// TwinCAT 3 PLC project xPPU_Lib
// Title: xPPU
// Company: Jan Wilch
// ProjectVersion: 1.0.0
// ProgramVersion: 3.1.4026.11
// libraries:
//   Tc2_Standard, * (Beckhoff Automation GmbH)
//   Tc2_System, * (Beckhoff Automation GmbH)
//   Tc3_Module, * (Beckhoff Automation GmbH)
//   [Resi4MPM], * (Jan Wilch)
// project tree:
//   03_ControlPrimitives/Carrier/Crane/ Crane_MoveBase.TcPOU, Crane_MoveToLSC.TcPOU, Crane_MoveToStack.TcPOU, Crane_MoveToStamp.TcPOU, Crane_PickPutBase.TcPOU, Crane_PickUpWP.TcPOU, Crane_PutDownWP.TcPOU
//   03_ControlPrimitives/Carrier/PickAlpha/ PicAlpha_MoveBase.TcPOU, PicAlpha_MoveToPos1.TcPOU, PicAlpha_MoveToPos2.TcPOU, PicAlpha_MoveToPos3.TcPOU, PicAlpha_MoveToPos4.TcPOU, PicAlpha_PickUpWP.TcPOU, PicAlpha_PutDownWP.TcPOU
//   03_ControlPrimitives/Conveyor/LSC/ LSC_MoveWorkpiece_Base.TcPOU, LSC_SearchWorkpiece.TcPOU, LSC_TransferWorkpieceTo_PAC.TcPOU, LSC_TransferWorkpieceTo_RampEnd.TcPOU, LSC_TransferWorkpieceTo_RampMid.TcPOU, LSC_TransferWorkpieceTo_RampStart.TcPOU
//   03_ControlPrimitives/Conveyor/PAC/ PAC_MoveWorkpiece_Base.TcPOU, PAC_TransferWorkpieceTo_PSEnd.TcPOU, PAC_TransferWorkpieceTo_PSStart.TcPOU, PAC_TransferWorkpieceTo_SSC.TcPOU
//   03_ControlPrimitives/Conveyor/RFC/ RFC_MoveWorkpiece_Base.TcPOU, RFC_TransferWorkpieceTo_LSC.TcPOU, RFC_TransferWorkpieceTo_PSEnd.TcPOU
//   03_ControlPrimitives/Conveyor/SSC/ SSC_MoveWorkpiece_Base.TcPOU, SSC_TransferWorkpieceTo_PSStart.TcPOU, SSC_TransferWorkpieceTo_RampEnd.TcPOU, SSC_TransferWorkpieceTo_RFC.TcPOU
//   03_ControlPrimitives/Generic/ Delay.TcPOU, ForceProcessVariable.TcPOU, IndicateActivity.TcPOU
//   03_ControlPrimitives/Stack/ Stack_ProvideWorkpiece.TcPOU
//   03_ControlPrimitives/Stamp/ Stamp_StampWorkpiece.TcPOU
//   04_HardwareObservation/ ObserveCrane.TcPOU, ObserveLSC.TcPOU, ObservePAC.TcPOU, ObservePicAlpha.TcPOU, ObserveRFC.TcPOU, ObserveSSC.TcPOU, ObserveStack.TcPOU, ObserveStamp.TcPOU, xPPUProduct.TcPOU
//   05_HardwareControl/ControlModule/ BaseComponent.TcPOU, Motor.TcPOU
//   05_HardwareControl/ControlModule/Gen/ ActivityIndicator.TcPOU
//   05_HardwareControl/ControlModule/Grippers/ BaseGripper.TcPOU, VacuumGripper.TcPOU
//   05_HardwareControl/ControlModule/Pushers/ BaseCylinder.TcPOU, BistableCylinder.TcPOU, MonostableCylinder.TcPOU, Switch.TcPOU
//   05_HardwareControl/ControlModule/Sensors/ InductiveSensor.TcPOU, OpticalSensor.TcPOU, PresenceSensor.TcPOU, PressureSensor.TcPOU, WeightSensor.TcPOU
//   05_HardwareControl/ControlModule/Valves/ PropotionalValve.TcPOU
//   05_HardwareControl/DUTs/ ActuatorConfiguration.TcDUT, BaseConfiguration.TcDUT, ConveyorConfiguration.TcDUT, ConveyorOutput.TcDUT, EWPMaterial.TcDUT, EWPWeight.TcDUT, MotorOutput.TcDUT, RampConfiguration.TcDUT, SensorConfiguration.TcDUT, SensorOutput.TcDUT
//   05_HardwareControl/EquipmentModule/Carriers/ BaseCarrier.TcPOU, Crane.TcPOU, PicAlpha.TcPOU
//   05_HardwareControl/EquipmentModule/Conveyors/ Conveyor.TcPOU, LargeSortingConveyor.TcPOU, PicAlphaConveyor.TcPOU, RefeedingConveyor.TcPOU, SmallSortingConveyor.TcPOU
//   05_HardwareControl/EquipmentModule/Ramps/ Ramp.TcPOU
//   05_HardwareControl/EquipmentModule/Stacks/ Stack.TcPOU
//   05_HardwareControl/EquipmentModule/Stamps/ Stamp.TcPOU
//   05_HardwareControl/Interfaces/ ITF_AnalogSensor.TcIO, ITF_BinarySensor.TcIO, ITF_Cylinder.TcIO
//   98_NamingEnums/ EAlarms.TcDUT, EOperatingModes.TcDUT, EPrimitives.TcDUT, EProcessVariables.TcDUT, EProducts.TcDUT, EProductTypes.TcDUT, ESequences.TcDUT, EStampStates.TcDUT
//   99_ExtrafunctionalImpl/ PanelManager.TcPOU, ErrorManager.TcPOU, FC_InitAlarmTexts.TcPOU, MachineModes.TcPOU
//   GVLs/ HMI_Texts.TcGVL
// real-time tasks:
//   TASK PlcTask: cycle T#10ms, priority 20, ADS port 350
//   TASK PlcTask1: cycle T#10ms, priority 23, ADS port 351
//   TASK PlcTask2: cycle T#10ms, priority 22, ADS port 352
//   TASK PlcTask3: cycle T#10ms, priority 21, ADS port 353
// I/O:
//   DEVICE Device (EtherCAT), AmsNetId 192.168.82.13.3.1
//     Term 84 (EK1200) [EK1200-5000 EtherCAT Netzteil (2A E-Bus)]
//       Klemme 2 (EK1110) [EK1110 EtherCAT-Verlängerung]
//     BK1 (EK1100) [EK1100 EtherCAT-Koppler (2A E-Bus)]
//       1.2 (EL1004) [EL1004 4K. Dig. Eingang 24V, 3ms]
//       1.3 (EL1004) [EL1004 4K. Dig. Eingang 24V, 3ms]
//       1.4 (EL1004) [EL1004 4K. Dig. Eingang 24V, 3ms]
//       1.5 (EL1004) [EL1004 4K. Dig. Eingang 24V, 3ms]
//       1.6 (EL2004) [EL2004 4K. Dig. Ausgang 24V, 0.5A]
//       1.9 (EL2004) [EL2004 4K. Dig. Ausgang 24V, 0.5A]
//       1.10 (EL2004) [EL2004 4K. Dig. Ausgang 24V, 0.5A]
//       1.11 (EL2004) [EL2004 4K. Dig. Ausgang 24V, 0.5A]
//       1.12 (EL1004) [EL1004 4K. Dig. Eingang 24V, 3ms]
//       1.13 (EL3162) [EL3162 2K. Ana. Eingang 0-10V]
//       1.14 (EL9011) [EL9011 Endklemme]
//     BK2&3 (EK1100) [EK1100 EtherCAT-Koppler (2A E-Bus)]
//       2&3.2 (EL1004) [EL1004 4K. Dig. Eingang 24V, 3ms]
//       2&3.3 (EL1004) [EL1004 4K. Dig. Eingang 24V, 3ms]
//       2&3.4 (EL1004) [EL1004 4K. Dig. Eingang 24V, 3ms]
//       2&3.5 (EL1004) [EL1004 4K. Dig. Eingang 24V, 3ms]
//       2&3.6 (EL1004) [EL1004 4K. Dig. Eingang 24V, 3ms]
//       2&3.7 (EL1004) [EL1004 4K. Dig. Eingang 24V, 3ms]
//       2&3.10 (EL2004) [EL2004 4K. Dig. Ausgang 24V, 0.5A]
//       2&3.11 (EL2004) [EL2004 4K. Dig. Ausgang 24V, 0.5A]
//       2&3.12 (EL2004) [EL2004 4K. Dig. Ausgang 24V, 0.5A]
//       2&3.13 (EL2004) [EL2004 4K. Dig. Ausgang 24V, 0.5A]
//       2&3.14 (EL1004) [EL1004 4K. Dig. Eingang 24V, 3ms]
//       2&3.16 (EL4102) [EL4102 2K. Ana. Ausgang 0-10V]
//       2&3.17 (EL4102) [EL4102 2K. Ana. Ausgang 0-10V]
//       2&3.18 (EL9011) [EL9011 Endklemme]
//     BK4 (EK1100) [EK1100 EtherCAT-Koppler (2A E-Bus)]
//       4.2 (EL1808) [EL1808 8K. Dig. Eingang 24V, 3ms]
//       4.3 (EL1004) [EL1004 4K. Dig. Eingang 24V, 3ms]
//       4.4 (EL1004) [EL1004 4K. Dig. Eingang 24V, 3ms]
//       4.5 (EL1004) [EL1004 4K. Dig. Eingang 24V, 3ms]
//       4.6 (EL1004) [EL1004 4K. Dig. Eingang 24V, 3ms]
//       4.7 (EL1004) [EL1004 4K. Dig. Eingang 24V, 3ms]
//       4.8 (EL3064) [EL3064 4K.Ana. Eingang 0-10V]
//       4.9 (EL3064) [EL3064 4K.Ana. Eingang 0-10V]
//       4.10 (EL3164) [EL3164 4K. Ana. Eingang 0-10V]
//       4.11 (EL3054) [EL3054 4K.Ana. Eingang 4-20mA]
//       Klemme 90 (EL3058) [EL3058 8K. Ana. Eingang 4-20mA]
//       4.13 (EL2004) [EL2004 4K. Dig. Ausgang 24V, 0.5A]
//       4.14 (EL2004) [EL2004 4K. Dig. Ausgang 24V, 0.5A]
//       4.15 (EL9011) [EL9011 Endklemme]
//     BK5 (EK1100) [EK1100 EtherCAT Coupler (2A E-Bus)]
//       5.2 (EL1008) [EL1008 8Ch. Dig. Input 24V, 3ms]
//       5.3 (EL5152) [EL5152 2Ch. Inc. Encoder]
//       5.6 (EL2008) [EL2008 8Ch. Dig. Output 24V, 0.5A]
//       5.7 (EL4102) [EL4102 2Ch. Ana. Output 0-10V]
//       5.8 (EL9011) [EL9011 End Terminal]
//     BK6 (EK1100) [EK1100 EtherCAT Coupler (2A E-Bus)]
//       6.2 (EL3062) [EL3062 2Ch. Ana. Input 0-10V]
//       6.3 (EL6224) [EL6224 (IO Link Master)]
//       6.4 (EL9011) [EL9011 End Terminal]
//     BK7 (EK1100) [EK1100 EtherCAT Coupler (2A E-Bus)]
//       7.2 (EL1004) [EL1004 4Ch. Dig. Input 24V, 3ms]
//       7.5 (EL2004) [EL2004 4Ch. Dig. Output 24V, 0.5A]
//       7.8 (EL6224) [EL6224 (IO Link Master)]
//       7.9 (EL9011) [EL9011 End Terminal]
//     BK8 (EK1100) [EK1100 EtherCAT Coupler (2A E-Bus)]
//       8.2 (EL1008) [EL1008 8Ch. Dig. Input 24V, 3ms]
//       8.3 (EL1004) [EL1004 4Ch. Dig. Input 24V, 3ms]
//       8.4 (EL3062) [EL3062 2Ch. Ana. Input 0-10V]
//       8.5 (EL2004) [EL2004 4Ch. Dig. Output 24V, 0.5A]
//       8.8 (EL2008) [EL2008 8Ch. Dig. Output 24V, 0.5A]
//       8.9 (EL2004) [EL2004 4Ch. Dig. Output 24V, 0.5A]
//       Term 114 (EL1808) [EL1808 8Ch. Dig. Input 24V, 3ms]
//       8.10 (EL9011) [EL9011 End Terminal]
//     BK9 (EK1100) [EK1100 EtherCAT Coupler (2A E-Bus)]
//       9.2 (EL1004) [EL1004 4Ch. Dig. Input 24V, 3ms]
//       9.3 (EL5152) [EL5152 2Ch. Inc. Encoder]
//       9.6 (EL2004) [EL2004 4Ch. Dig. Output 24V, 0.5A]
//       9.7 (EL4102) [EL4102 2Ch. Ana. Output 0-10V]
//       9.8 (EL9011) [EL9011 End Terminal]
//     BK10 (EK1100) [EK1100 EtherCAT Coupler (2A E-Bus)]
//       10.2 (EL1004) [EL1004 4Ch. Dig. Input 24V, 3ms]
//       10.3 (EL5152) [EL5152 2Ch. Inc. Encoder]
//       10.6 (EL2004) [EL2004 4Ch. Dig. Output 24V, 0.5A]
//       10.7 (EL4102) [EL4102 2Ch. Ana. Output 0-10V]
//       10.8 (EL9011) [EL9011 End Terminal]
//     BK11 (EK1100) [EK1100 EtherCAT Coupler (2A E-Bus)]
//       11.2 (EL1004) [EL1004 4Ch. Dig. Input 24V, 3ms]
//       11.3 (EL3064) [EL3064 4Ch. Ana. Input 0-10V]
//       11.6 (EL2004) [EL2004 4Ch. Dig. Output 24V, 0.5A]
//       11.7 (EL9011) [EL9011 End Terminal]

// ---- 05_HardwareControl/DUTs/ActuatorConfiguration.TcDUT
TYPE ActuatorConfiguration EXTENDS BaseConfiguration:
STRUCT
	//Output
	sPusherType : STRING;
	iPusherPosition : DINT;
END_STRUCT
END_TYPE

// ---- 05_HardwareControl/DUTs/BaseConfiguration.TcDUT
TYPE BaseConfiguration :
STRUCT
	sName : STRING;
	sOutputDescription : STRING;
	sMountingPoint : STRING;
END_STRUCT
END_TYPE

// ---- 05_HardwareControl/DUTs/ConveyorConfiguration.TcDUT
TYPE ConveyorConfiguration :
STRUCT
	iNumSensor : DINT;
	iNumRamp : DINT;
	iNumPusher : DINT;
END_STRUCT
END_TYPE

// ---- 05_HardwareControl/DUTs/ConveyorOutput.TcDUT
TYPE ConveyorOutput :
STRUCT
	SensorDataOutput : ARRAY[0..10] OF SensorOutput;
	SensorNum : DINT;
	//Ramps
	RampDataOutput : ARRAY[0..5] OF SensorOutput;
	RampNum : DINT;
	//Pushers
	PusherOut : ARRAY[0..10] OF SensorOutput;
	PusherNum : DINT;
	//Motor Output
	MotorOutput : MotorOutput;
END_STRUCT
END_TYPE

// ---- 05_HardwareControl/DUTs/EWPMaterial.TcDUT
{attribute 'qualified_only'}
{attribute 'strict'}
TYPE EWPMaterial :
(
	black := 1,
	white := 2,
	metallic :=3,
	undetermined :=4,
	enum_member := 0
);
END_TYPE

// ---- 05_HardwareControl/DUTs/EWPWeight.TcDUT
{attribute 'qualified_only'}
{attribute 'strict'}
TYPE EWPWeight :
(
	light :=1,
	medium := 2,
	heavy := 3,
	undetermined :=4,
	enum_member := 0
);
END_TYPE

// ---- 05_HardwareControl/DUTs/MotorOutput.TcDUT
TYPE MotorOutput :
STRUCT
	ConveyorForward : BOOL;
	ConveyorBackward : BOOL;
	ConveyorStop : BOOL;
	ConveyorSpeed : UDINT;
END_STRUCT
END_TYPE

// ---- 05_HardwareControl/DUTs/RampConfiguration.TcDUT
TYPE RampConfiguration EXTENDS BaseConfiguration:
STRUCT
END_STRUCT
END_TYPE

// ---- 05_HardwareControl/DUTs/SensorConfiguration.TcDUT
TYPE SensorConfiguration EXTENDS BaseConfiguration:
STRUCT
	sReturnType : STRING;
	sType : STRING;
	sSensPosition : STRING;
	iSensIndex : DINT;
END_STRUCT
END_TYPE

// ---- 05_HardwareControl/DUTs/SensorOutput.TcDUT
TYPE SensorOutput :
STRUCT
	SensorName : STRING;
	SensorActive : BOOL;
	
	OutputType : STRING;
	OutputDescription : STRING;
	//OutputINT : INT;
	OutputBOOL : BOOL;
	//OutputREAL : REAL;
END_STRUCT
END_TYPE

// ---- 98_NamingEnums/EAlarms.TcDUT
{attribute 'qualified_only'}
{attribute 'strict'}
TYPE EAlarms :
(
	none := 0,
	initialized := 1,
	did_execute := 2,
	sequence_failed := 3,
	stopping := 4,
	aborting := 5,
	stopped := 6
) UINT;
END_TYPE

// ---- 98_NamingEnums/EOperatingModes.TcDUT
{attribute 'qualified_only'}
{attribute 'strict'}
{attribute 'to_string'}
// TODO - adapt to PackML (?)
TYPE EOperatingModes :
(
	none := 0,
	init := 1,
	automatic := 2,
	manual := 3,
	recovering := 4,
	shutting_down := 5,
	shutdown := 6,
	custom_sequence := 7
) UINT;
END_TYPE

// ---- 98_NamingEnums/EPrimitives.TcDUT
{attribute 'qualified_only'}
{attribute 'strict'}
TYPE EPrimitives :
(
	empty := 0,
	
	Crane_MoveToStack := 01,
	Crane_MoveToLSC := 02,
	Crane_MoveToStamp := 03,
	Crane_PickUpWP := 04,
	Crane_PutDownWP := 05,
	
	Stamp_StampWorkpiece := 10,
	
	Stack_ProvideWorkpiece := 20,
	
	LSC_TransferWorkpieceTo_RampStart := 30,
	LSC_TransferWorkpieceTo_RampMid := 31,
	LSC_TransferWorkpieceTo_RampEnd := 32,
	LSC_TransferWorkpieceTo_PAC := 33,
	LSC_SearchWorkpiece := 35,
	
	PAC_TransferWorkpieceTo_PSStart := 40,
	PAC_TransferWorkpieceTo_PSEnd := 41,
	PAC_TransferWorkpieceTo_SSC := 42,
	
	PicAlpha_MoveToPos1 := 50,
	PicAlpha_MoveToPos2 := 51,
	PicAlpha_MoveToPos3 := 52,
	PicAlpha_MoveToPos4 := 53,
	PicAlpha_PickUpWP := 54,
	PicAlpha_PutDownWp := 55,
	
	SSC_TransferWorkpieceTo_PSStart := 60,
	SSC_TransferWorkpieceTo_RampEnd := 61,
	SSC_TransferWorkpieceTo_RFC := 62,
	
	RFC_TransferWorkpieceTo_PSEnd := 70,
	RFC_TransferWorkpieceTo_LSC := 71,
	
	Gen_Delay := 90,
	Gen_IndicateActive_Crane := 91,
	Gen_IndicateActive_Stack := 92,
	Gen_IndicateActive_Stamp := 93,
	Gen_IndicateActive_LSC := 94,
	Gen_ForceVariable_Crane := 95,
	Gen_ForceVariable_Stack := 96,
	Gen_ForceVariable_Stamp := 97,
	Gen_ForceVariable_LSC := 98
) UINT;
END_TYPE

// ---- 98_NamingEnums/EProcessVariables.TcDUT
{attribute 'qualified_only'}
{attribute 'to_string'}
TYPE EProcessVariables :
(
	none := 0,
	
	OpMode_Stack := 1,
	OpMode_Crane := 2,
	OpMode_Stamp := 3,
	OpMode_LSC := 4,
	
	Stack_WorkpieceAvailable := 10,
	Stack_ProductType := 11,
	Stack_ProductStamped := 12,
	Stack_CylinderExtended := 13,
	Stack_CylinderRetracted := 14,
	
	Crane_AtStack := 20,
	Crane_AtStamp := 21,
	Crane_AtLSC := 22,
	Crane_HoldingWorkpiece := 23,
	Crane_CylinderExtended := 24,
	Crane_CylinderRetracted := 25,
	Crane_Angle := 26,
	Crane_ProductType := 27,
	Crane_ProductStamped := 28,
	
	// the state of a workpiece at the stamp: 0=no workpiece, 1=workpiece received, 2=workpiece processed, 3=busy
	Stamp_WorkpieceState := 30,
	Stamp_WPAtStamp := 31,
	Stamp_ProductType := 32,
	Stamp_ProductStamped := 33,
	Stamp_StamperExtended := 34,
	Stamp_StamperRetracted := 35,
	Stamp_SliderExtended := 36,
	Stamp_SliderRetracted := 37,
	
	LSC_WorkpieceAtEntry := 40,
	LSC_SwitchExtended := 41,
	LSC_SwitchRetracted := 42,
	LSC_WPAtRampStart := 43,
	LSC_WPAtRampMiddle := 44,
	LSC_WPAtRampEnd := 45,
	LSC_WPAtInductiveSensorEnd := 48,
	LSC_ProductType := 49,
	LSC_ProductStamped := 50,
	LSC_RampStartWPCount := 51,
	LSC_RampMiddleWPCount := 52,
	LSC_RampEndWPCount := 53,
	
	PAC_WPAtStart := 60,
	PAC_WPAtEnd := 61,
	PAC_SwitchExtended := 62,
	PAC_SwitchRetracted := 63,
	PAC_WPNumber := 64,
	PAC_ProductType_1 := 65,
	PAC_ProductType_2 := 66,
	PAC_ProductType_3 := 67,
	
	PicAlpha_AtPos1 := 70,
	PicAlpha_AtPos2 := 71,
	PicAlpha_AtPos3 := 72,
	PicAlpha_AtPos4 := 73,
	PicAlpha_HoldingWorkpiece := 74,
	PicAlpha_CylinderExtended := 75,
	PicAlpha_CylinderRetracted := 76,
	PicAlpha_Distance := 77,
	PicAlpha_ProductType := 78,
	
	SSC_SwitchExtended := 80,
	SSC_SwitchRetracted := 81,
	SSC_WPAtStart := 82,
	SSC_WPLightAtMiddle := 83,
	SSC_WPMetalAtMiddle := 84,
	SSC_WPAtEnd := 85,
	SSC_WPAtRampEnd := 86,
	SSC_ProductType_1 := 87,
	SSC_ProductType_2 := 88,
	SSC_RampWPCount := 89,
	
	RFC_SwitchExtended := 90,
	RFC_SwitchRetracted := 91,
	RFC_WPAtStart := 92,
	RFC_WPAtEnd := 93,
	RFC_ProductType_1 := 94,
	RFC_ProductType_2 := 95,
	
	// Stack panel
	Pnl_Stack_Start := 100,
	Pnl_Stack_Mode := 101,
	Pnl_Stack_EStop := 102,
	// LSC panel
	Pnl_LSC_Start := 103,
	Pnl_LSC_Mode := 104,
	Pnl_LSC_EStop := 105,
	// Stamp panel
	Pnl_Stamp_Start := 106,
	Pnl_Stamp_Mode := 107,
	Pnl_Stamp_EStop := 108,
	// Light barrier safety panel
	Pnl_LightBarrier_Start := 109,
	Pnl_LightBarrier_Stop := 110,
	Pnl_LightBarrier_Mode := 111,
	Pnl_LightBarrier_EStop := 112,
	Pnl_LightBarrier_Reset := 113,
	// Door safety panel
	Pnl_Door_Start := 114,
	Pnl_Door_Stop := 115,
	Pnl_Door_Mode := 116,
	Pnl_Door_EStop := 117,	// currently not connected to PLC
	Pnl_Door_Reset := 118,
	
	Test_CraneFree := 120,
	Test_StampFree := 121,
	Test_StackFree := 122,
	Test_LSCFree := 123
) UINT;
END_TYPE

// ---- 98_NamingEnums/EProducts.TcDUT
{attribute 'qualified_only'}
{attribute 'strict'}
TYPE EProducts :
(
	none := 0,
	stack_product := 1,
	crane_product := 2,
	stamp_product := 3,
	LSC_product := 4,
	PAC_product1 := 5,
	PAC_product2 := 6,
	PAC_product3 := 7,
	PicAlpha_product := 8,
	RFC_product1 := 9,
	RFC_product2 := 10,
	SSC_product1 := 11,
	SSC_product2 := 12
) UINT;
END_TYPE

// ---- 98_NamingEnums/EProductTypes.TcDUT
{attribute 'qualified_only'}
TYPE EProductTypes :
(
	none := 0,
	unknown := 1,
	
	white := 2,
	black := 3,
	metal := 4
) UINT;
END_TYPE

// ---- 98_NamingEnums/ESequences.TcDUT
{attribute 'qualified_only'}
{attribute 'strict'}
TYPE ESequences :
(
	empty := 0,
	sample_sequence := 1
) UINT;
END_TYPE

// ---- 98_NamingEnums/EStampStates.TcDUT
{attribute 'qualified_only'}
{attribute 'strict'}
TYPE EStampStates :
(
	none := 0,
	unpressed := 1,
	pressed := 2,
	busy := 3
) UINT;
END_TYPE

// ---- GVLs/HMI_Texts.TcGVL
{attribute 'qualified_only'}
VAR_GLOBAL
	AlarmTexts: ARRAY [0..999] OF STRING;
END_VAR

// ---- 05_HardwareControl/Interfaces/ITF_AnalogSensor.TcIO
INTERFACE ITF_AnalogSensor

PROPERTY Value : INT
GET
END_GET
END_PROPERTY

END_INTERFACE

// ---- 05_HardwareControl/Interfaces/ITF_BinarySensor.TcIO
INTERFACE ITF_BinarySensor

PROPERTY Value : BOOL
GET
END_GET
END_PROPERTY

END_INTERFACE

// ---- 05_HardwareControl/Interfaces/ITF_Cylinder.TcIO
INTERFACE ITF_Cylinder

PROPERTY Extended : BOOL
GET
END_GET
END_PROPERTY

METHOD METH_Extend : BOOL
END_METHOD

METHOD METH_Retract : BOOL
END_METHOD

PROPERTY Retracted : BOOL
GET
END_GET
END_PROPERTY

END_INTERFACE

// ---- 03_ControlPrimitives/Carrier/Crane/Crane_MoveBase.TcPOU
FUNCTION_BLOCK ABSTRACT Crane_MoveBase EXTENDS ControlPrimitiveBase
VAR_INPUT
END_VAR
VAR_OUTPUT
END_VAR
VAR
	m_ptrCrane: POINTER TO Crane;
END_VAR

SUPER^();

METHOD Abort : BOOL
VAR_INPUT
END_VAR
m_ptrCrane^.METH_CarrierStop();
Abort := TRUE;
END_METHOD

PROPERTY ABSTRACT AtTarget : BOOL
GET
END_GET
END_PROPERTY

(* Execution logic of this Control Primitive. *)
METHOD PROTECTED ExecuteInternal : BOOL
VAR_INPUT
	i_params	: Resi4MPM.ParameterSet;
END_VAR
VAR
	angle: REAL;
	diff: REAL;
END_VAR
angle := m_st^.GetNumeric(EProcessVariables.Crane_Angle);
diff := TargetAngle - angle;

IF AtTarget THEN
	m_ptrCrane^.METH_CarrierStop();
	ExecuteInternal := TRUE;
ELSIF diff < 0 THEN
	m_ptrCrane^.METH_CarrierTurnClockwise();
ELSE
	m_ptrCrane^.METH_CarrierTurnCounterClockwise();
END_IF
END_METHOD

PROPERTY ABSTRACT TargetAngle : UINT
GET
END_GET
END_PROPERTY

END_FUNCTION_BLOCK

// ---- 05_HardwareControl/EquipmentModule/Carriers/Crane.TcPOU
FUNCTION_BLOCK Crane EXTENDS BaseCarrier
VAR_INPUT
END_VAR
VAR_OUTPUT
	o_VacuumGripper: VacuumGripper;
	o_MonostableCylinder: MonostableCylinder;
END_VAR
VAR
	// Turning table
	m_PresenceSensorAtStack : PresenceSensor;
	m_PresenceSensorAtConveyor : PresenceSensor;
	m_PresenceSensorAtStamp : PresenceSensor;
END_VAR

PROPERTY AtConveyor : BOOL
GET
AtConveyor := m_PresenceSensorAtConveyor.Value;
END_GET
END_PROPERTY

PROPERTY AtStack : BOOL
GET
AtStack := m_PresenceSensorAtStack.Value;
END_GET
END_PROPERTY

PROPERTY AtStamp : BOOL
GET
AtStamp := m_PresenceSensorAtStamp.Value;
END_GET
END_PROPERTY

METHOD METH_CarrierStop : BOOL
VAR_INPUT
END_VAR
Motor.ACT_Stop();
END_METHOD

METHOD METH_CarrierTurnClockwise : BOOL
VAR_INPUT
END_VAR
Motor.ACT_TurnClockwise();
END_METHOD

METHOD METH_CarrierTurnCounterclockwise : BOOL
VAR_INPUT
END_VAR
Motor.ACT_TurnCounterclockwise();
END_METHOD

END_FUNCTION_BLOCK

// ---- 05_HardwareControl/EquipmentModule/Carriers/BaseCarrier.TcPOU
FUNCTION_BLOCK BaseCarrier EXTENDS BaseComponent
VAR_INPUT
END_VAR
VAR_OUTPUT
END_VAR
VAR
	Motor : Motor;
END_VAR

END_FUNCTION_BLOCK

// ---- 05_HardwareControl/ControlModule/BaseComponent.TcPOU
FUNCTION_BLOCK BaseComponent
VAR_INPUT
END_VAR
VAR_OUTPUT
END_VAR
VAR
END_VAR

END_FUNCTION_BLOCK

// ---- 05_HardwareControl/ControlModule/Motor.TcPOU
FUNCTION_BLOCK Motor
VAR_INPUT
	//Software
	Stopped : BOOL;
	TurningClockwise : BOOL;
	TurningCounterclockwise : BOOL;
END_VAR
VAR_OUTPUT	
	AI_Position AT %I*: UINT;
	AI_Speed AT %I*: UDINT;
END_VAR
VAR	
	//Hardware
	DO_TurnClockwise AT %Q* : BOOL;
	DO_TurnCounterclockwise AT %Q* : BOOL;	
END_VAR

ACTION ACT_Stop:
DO_TurnClockwise := FALSE;
DO_TurnCounterclockwise := FALSE;

Stopped := TRUE;
TurningClockwise := FALSE;
TurningCounterclockwise := FALSE;
END_ACTION

ACTION ACT_TurnClockwise:
DO_TurnClockwise := TRUE;
DO_TurnCounterclockwise := FALSE;

Stopped := FALSE;
TurningClockwise := TRUE;
TurningCounterclockwise := FALSE;
END_ACTION

ACTION ACT_TurnCounterclockwise:
DO_TurnClockwise := FALSE;
DO_TurnCounterclockwise := TRUE;

Stopped := FALSE;
TurningClockwise := FALSE;
TurningCounterclockwise := TRUE;
END_ACTION

END_FUNCTION_BLOCK

// ---- 05_HardwareControl/ControlModule/Grippers/VacuumGripper.TcPOU
FUNCTION_BLOCK VacuumGripper EXTENDS BaseGripper
VAR_INPUT
END_VAR
VAR_OUTPUT
END_VAR
VAR
	//Hardware
	DI_TakenIn AT %I* : BOOL;
	DO_VacuumOn AT %Q* : BOOL;
	// Only used by PickAlpha
	VacuumHit AT %Q* : BOOL;
END_VAR

METHOD METH_Intake : BOOL
VAR_INPUT
END_VAR
DO_VacuumOn := TRUE;
END_METHOD

METHOD METH_Release : BOOL
VAR_INPUT
END_VAR
DO_VacuumOn := FALSE;
END_METHOD

METHOD METH_VacuumHitOff : BOOL
VAR_INPUT
END_VAR
VacuumHit := FALSE;
END_METHOD

METHOD METH_VacuumHitOn : BOOL
VAR_INPUT
END_VAR
VacuumHit := TRUE;
END_METHOD

PROPERTY WPTaken : BOOL
GET
// TODO - connect input correctly (probably hardware issue)
WPTaken := DI_TakenIn;
//WPTaken := DO_VacuumOn;
END_GET
END_PROPERTY

END_FUNCTION_BLOCK

// ---- 05_HardwareControl/ControlModule/Grippers/BaseGripper.TcPOU
FUNCTION_BLOCK BaseGripper
VAR_INPUT
END_VAR
VAR_OUTPUT
END_VAR
VAR
END_VAR

END_FUNCTION_BLOCK

// ---- 05_HardwareControl/ControlModule/Pushers/MonostableCylinder.TcPOU
FUNCTION_BLOCK MonostableCylinder EXTENDS BaseCylinder
VAR_INPUT
END_VAR
VAR_OUTPUT
END_VAR
VAR
END_VAR

METHOD METH_Extend : BOOL
DO_Extend := TRUE;
END_METHOD

METHOD METH_Retract : BOOL
DO_Extend := FALSE;
END_METHOD

END_FUNCTION_BLOCK

// ---- 05_HardwareControl/ControlModule/Pushers/BaseCylinder.TcPOU
FUNCTION_BLOCK ABSTRACT BaseCylinder IMPLEMENTS ITF_Cylinder
VAR_INPUT
END_VAR
VAR_OUTPUT
END_VAR
VAR
	//Hardware
	DI_Extended AT %I* : BOOL;
	DI_Retracted AT %I* : BOOL;
	DO_Extend AT %Q* : BOOL;
	//NOT USED BUT USABLE	
	DI_BoundaryPressure AT %I* : BOOL;
	DI_BoundaryFlowPressure AT %I* : BOOL;
	AI_PressureSensor AT %I* : INT;
	AI_FlowPressure AT %I* : INT;
	AI_PositionTransmitter AT %I* : INT;
END_VAR

PROPERTY Extended : BOOL
GET
Extended := DI_Extended;
END_GET
END_PROPERTY

METHOD ABSTRACT METH_Extend : BOOL
END_METHOD

METHOD ABSTRACT METH_Retract : BOOL
END_METHOD

PROPERTY Retracted : BOOL
GET
Retracted := DI_Retracted;
END_GET
END_PROPERTY

END_FUNCTION_BLOCK

// ---- 05_HardwareControl/ControlModule/Sensors/PresenceSensor.TcPOU
FUNCTION_BLOCK PresenceSensor IMPLEMENTS ITF_BinarySensor
VAR_INPUT
END_VAR
VAR_OUTPUT
END_VAR
VAR
	DI_WPDetected AT %I* : BOOL;
END_VAR

PROPERTY Value : BOOL
GET
Value := DI_WPDetected;
END_GET
END_PROPERTY

END_FUNCTION_BLOCK

// ---- 03_ControlPrimitives/Carrier/Crane/Crane_MoveToLSC.TcPOU
FUNCTION_BLOCK Crane_MoveToLSC EXTENDS Crane_MoveBase
VAR_INPUT
END_VAR
VAR_OUTPUT
END_VAR
VAR
	// (EProcessVariables.Crane_CylinderRetracted = TRUE) AND ((EProcessVariables.Crane_HoldingWorkpiece = FALSE) OR ((EProcessVariables.LSC_ProductType = 0) AND ((EProcessVariables.RFC_ProductType_1 = 0) AND (EProcessVariables.RFC_ProductType_2 = 0))))
	m_compExpr1: ComparisonExpression(EProcessVariables.Crane_CylinderRetracted, EComparisonType.equals, EDataType.binary, TRUE, 0, '', TRUE);
	m_compExpr3: ComparisonExpression(EProcessVariables.Crane_HoldingWorkpiece, EComparisonType.equals, EDataType.binary, FALSE, 0, '', TRUE);
	m_compExpr5: ComparisonExpression(EProcessVariables.LSC_ProductType, EComparisonType.equals, EDataType.numeric, FALSE, 0, '', TRUE);
// 	m_compExpr7: ComparisonExpression(EProcessVariables.RFC_ProductType_1, EComparisonType.equals, EDataType.numeric, FALSE, 0, '', TRUE);
// 	m_compExpr9: ComparisonExpression(EProcessVariables.RFC_ProductType_2, EComparisonType.equals, EDataType.numeric, FALSE, 0, '', TRUE);
// 	m_boolExpr10: BoolExpression(m_compExpr7, EBoolOperation.and_op, m_compExpr9);
// 	m_boolExpr11: BoolExpression(m_compExpr5, EBoolOperation.and_op, m_boolExpr10);
// 	m_boolExpr12: BoolExpression(m_compExpr3, EBoolOperation.or_op, m_boolExpr11);
	m_boolExpr12: BoolExpression(m_compExpr3, EBoolOperation.or_op, m_compExpr5);
	m_precondition: BoolExpression(m_compExpr1, EBoolOperation.and_op, m_boolExpr12);
	
	// EProcessVariables.Crane_AtLSC = TRUE
	m_postcondition: ComparisonExpression(EProcessVariables.Crane_AtLSC, EComparisonType.equals, EDataType.binary, TRUE, 0, '', TRUE);
END_VAR

SUPER^();

PROPERTY AtTarget : BOOL
GET
AtTarget := m_ptrCrane^.AtConveyor;
END_GET
END_PROPERTY

METHOD FB_init : BOOL
VAR_INPUT
	bInitRetains : BOOL; // if TRUE, the retain variables are initialized (warm start / cold start)
	bInCopyCode : BOOL;  // if TRUE, the instance afterwards gets moved into the copy code (online change)
		
	i_ptrCrane: POINTER TO Crane;
END_VAR
m_ptrCrane := i_ptrCrane;

m_id := EPrimitives.Crane_MoveToLSC;
m_timeout := T#30S;

Precondition := m_precondition;
Postcondition := m_postcondition;
END_METHOD

PROPERTY TargetAngle : UINT
GET
TargetAngle := 90;
END_GET
END_PROPERTY

END_FUNCTION_BLOCK

// ---- 03_ControlPrimitives/Carrier/Crane/Crane_MoveToStack.TcPOU
FUNCTION_BLOCK Crane_MoveToStack EXTENDS Crane_MoveBase
VAR_INPUT
END_VAR
VAR_OUTPUT
END_VAR
VAR
	m_precondition: ComparisonExpression(EProcessVariables.Crane_CylinderRetracted, EComparisonType.equals, EDataType.binary, TRUE, 0, '', TRUE);
	
	// EProcessVariables.Crane_AtStack = TRUE
	m_postcondition: ComparisonExpression(EProcessVariables.Crane_AtStack, EComparisonType.equals, EDataType.binary, TRUE, 0, '', TRUE);
END_VAR

SUPER^();

PROPERTY AtTarget : BOOL
GET
AtTarget := m_ptrCrane^.AtStack;
END_GET
END_PROPERTY

METHOD FB_init : BOOL
VAR_INPUT
	bInitRetains : BOOL; // if TRUE, the retain variables are initialized (warm start / cold start)
	bInCopyCode : BOOL;  // if TRUE, the instance afterwards gets moved into the copy code (online change)
		
	i_ptrCrane: POINTER TO Crane;
END_VAR
m_ptrCrane := i_ptrCrane;

m_id := EPrimitives.Crane_MoveToStack;
m_timeout := T#30S;

Precondition := m_precondition;
Postcondition := m_postcondition;
END_METHOD

PROPERTY TargetAngle : UINT
GET
TargetAngle := 0;
END_GET
END_PROPERTY

END_FUNCTION_BLOCK

// ---- 03_ControlPrimitives/Carrier/Crane/Crane_MoveToStamp.TcPOU
FUNCTION_BLOCK Crane_MoveToStamp EXTENDS Crane_MoveBase
VAR_INPUT
END_VAR
VAR_OUTPUT
END_VAR
VAR
	// Crane_CylinderRetracted
	m_precondition: ComparisonExpression(EProcessVariables.Crane_CylinderRetracted, EComparisonType.equals, EDataType.binary, TRUE, 0, '', TRUE);
	
	// EProcessVariables.Crane_AtStamp = TRUE
	m_postcondition: ComparisonExpression(EProcessVariables.Crane_AtStamp, EComparisonType.equals, EDataType.binary, TRUE, 0, '', TRUE);
END_VAR

SUPER^();

PROPERTY AtTarget : BOOL
GET
AtTarget := m_ptrCrane^.AtStamp;
END_GET
END_PROPERTY

METHOD FB_init : BOOL
VAR_INPUT
	bInitRetains : BOOL; // if TRUE, the retain variables are initialized (warm start / cold start)
	bInCopyCode : BOOL;  // if TRUE, the instance afterwards gets moved into the copy code (online change)
		
	i_ptrCrane: POINTER TO Crane;
END_VAR
m_ptrCrane := i_ptrCrane;

m_id := EPrimitives.Crane_MoveToStamp;
m_timeout := T#30S;

Precondition := m_precondition;
Postcondition := m_postcondition;
END_METHOD

PROPERTY TargetAngle : UINT
GET
TargetAngle := 180;
END_GET
END_PROPERTY

END_FUNCTION_BLOCK

// ---- 03_ControlPrimitives/Carrier/Crane/Crane_PickPutBase.TcPOU
FUNCTION_BLOCK ABSTRACT Crane_PickPutBase EXTENDS ControlPrimitiveBase
VAR
	m_ptrCrane: POINTER TO Crane;
END_VAR

SUPER^();

METHOD PROTECTED ShiftProduct : BOOL
VAR_INPUT
	i_isIncoming: BOOL;
END_VAR
IF m_ptrCrane^.AtStack THEN
	IF i_isIncoming THEN
		ShiftProduct := m_st^.ShiftProduct(EProducts.stack_product, EProducts.crane_product);
	ELSE
		ShiftProduct := m_st^.ShiftProduct(EProducts.crane_product, EProducts.stack_product);
	END_IF
ELSIF m_ptrCrane^.AtConveyor THEN
	IF i_isIncoming THEN
		ShiftProduct := m_st^.ShiftProduct(EProducts.LSC_product, EProducts.crane_product);
	ELSE
		ShiftProduct := m_st^.ShiftProduct(EProducts.crane_product, EProducts.LSC_product);
	END_IF
ELSIF m_ptrCrane^.AtStamp THEN
	IF i_isIncoming THEN
		ShiftProduct := m_st^.ShiftProduct(EProducts.stamp_product, EProducts.crane_product);
	ELSE
		ShiftProduct := m_st^.ShiftProduct(EProducts.crane_product, EProducts.stamp_product);
	END_IF
END_IF
END_METHOD

END_FUNCTION_BLOCK

// ---- 03_ControlPrimitives/Carrier/Crane/Crane_PickUpWP.TcPOU
FUNCTION_BLOCK Crane_PickUpWP EXTENDS Crane_PickPutBase
VAR_INPUT
END_VAR
VAR_OUTPUT
END_VAR
VAR
	m_step: INT := 0;
	m_timer: TON;
	
	// (EProcessVariables.Crane_HoldingWorkpiece = FALSE) AND (EProcessVariables.Crane_CylinderRetracted = TRUE)
	m_compExpr55: ComparisonExpression(EProcessVariables.Crane_HoldingWorkpiece, EComparisonType.equals, EDataType.binary, FALSE, 0, '', TRUE);
	m_compExpr57: ComparisonExpression(EProcessVariables.Crane_CylinderRetracted, EComparisonType.equals, EDataType.binary, TRUE, 0, '', TRUE);
	m_precondition: BoolExpression(m_compExpr55, EBoolOperation.and_op, m_compExpr57);
	
	// (Crane_HoldingWorkpiece AND Crane_CylinderRetracted) AND ((Crane_AtStack AND Stack_ProductType = 0.0) OR ((Crane_AtStamp AND Stamp_ProductType = 0.0) OR (Crane_AtLSC AND LSC_ProductType = 0.0)))
	m_compExp224: ComparisonExpression(EProcessVariables.Crane_HoldingWorkpiece, EComparisonType.equals, EDataType.binary, TRUE, 0, '', TRUE);
	m_compExp226: ComparisonExpression(EProcessVariables.Crane_CylinderRetracted, EComparisonType.equals, EDataType.binary, True, 0, '', TRUE);
	m_boolExp222: BoolExpression(m_compExp224, EBoolOperation.and_op, m_compExp226);
	m_compExp232: ComparisonExpression(EProcessVariables.Crane_AtStack, EComparisonType.equals, EDataType.binary, True, 0, '', TRUE);
	m_compExp234: ComparisonExpression(EProcessVariables.Stack_ProductType, EComparisonType.equals, EDataType.numeric, FALSE, 0.0, '', TRUE);
	m_boolExp230: BoolExpression(m_compExp232, EBoolOperation.and_op, m_compExp234);
	m_compExp244: ComparisonExpression(EProcessVariables.Crane_AtStamp, EComparisonType.equals, EDataType.binary, True, 0, '', TRUE);
	m_compExp246: ComparisonExpression(EProcessVariables.Stamp_ProductType, EComparisonType.equals, EDataType.numeric, FALSE, 0.0, '', TRUE);
	m_boolExp242: BoolExpression(m_compExp244, EBoolOperation.and_op, m_compExp246);
	m_compExp259: ComparisonExpression(EProcessVariables.Crane_AtLSC, EComparisonType.equals, EDataType.binary, True, 0, '', TRUE);
	m_compExp261: ComparisonExpression(EProcessVariables.LSC_ProductType, EComparisonType.equals, EDataType.numeric, FALSE, 0.0, '', TRUE);
	m_boolExp257: BoolExpression(m_compExp259, EBoolOperation.and_op, m_compExp261);
	m_boolExp241: BoolExpression(m_boolExp242, EBoolOperation.or_op, m_boolExp257);
	m_boolExp229: BoolExpression(m_boolExp230, EBoolOperation.or_op, m_boolExp241);
	m_postcondition: BoolExpression(m_boolExp222, EBoolOperation.and_op, m_boolExp229);
END_VAR

SUPER^();

METHOD Abort : BOOL
VAR_INPUT
END_VAR
m_ptrCrane^.o_MonostableCylinder.METH_Retract();
IF m_ptrCrane^.o_VacuumGripper.WPTaken THEN
	m_ptrCrane^.o_VacuumGripper.METH_Intake();
ELSE
	m_ptrCrane^.o_VacuumGripper.METH_Release();
END_IF
Abort := TRUE;
END_METHOD

(* Execution logic of this Control Primitive. *)
METHOD PROTECTED  ExecuteInternal : BOOL
VAR_INPUT
	i_params: ParameterSet;
END_VAR
CASE m_step OF
	0:	// extend
		m_ptrCrane^.o_MonostableCylinder.METH_Extend();
		IF m_ptrCrane^.o_MonostableCylinder.Extended THEN
			m_step := 1;
		END_IF
	
	1:	// grip
		m_ptrCrane^.o_VacuumGripper.METH_Intake();
		m_timer(IN := TRUE, PT := T#1S);
		IF m_timer.Q THEN
			m_timer(IN := FALSE);
			m_step := 2;
		END_IF
	
	2: // shift register
		IF ShiftProduct(TRUE) THEN
			m_step := 3;
		END_IF
	
	3:	// retract
		m_ptrCrane^.o_MonostableCylinder.METH_Retract();
		IF m_ptrCrane^.o_MonostableCylinder.Retracted THEN
			m_step := 0;
			ExecuteInternal := TRUE;
		END_IF	
END_CASE
END_METHOD

METHOD FB_init : BOOL
VAR_INPUT
	bInitRetains : BOOL; // if TRUE, the retain variables are initialized (warm start / cold start)
	bInCopyCode : BOOL;  // if TRUE, the instance afterwards gets moved into the copy code (online change)
	
	i_ptrCrane: POINTER TO Crane;
END_VAR
m_ptrCrane := i_ptrCrane;

m_id := EPrimitives.Crane_PickUpWP;
m_timeout := T#10S;

Precondition := m_precondition;
Postcondition := m_postcondition;
END_METHOD

END_FUNCTION_BLOCK

// ---- 03_ControlPrimitives/Carrier/Crane/Crane_PutDownWP.TcPOU
FUNCTION_BLOCK Crane_PutDownWP EXTENDS Crane_PickPutBase
VAR_INPUT
END_VAR
VAR_OUTPUT
END_VAR
VAR
	m_step: INT := 0;
	m_timer: TON;

	// (EProcessVariables.Crane_HoldingWorkpiece = TRUE) AND (EProcessVariables.Crane_CylinderRetracted = TRUE)
	m_compExpr65: ComparisonExpression(EProcessVariables.Crane_HoldingWorkpiece, EComparisonType.equals, EDataType.binary, TRUE, 0, '', TRUE);
	m_compExpr67: ComparisonExpression(EProcessVariables.Crane_CylinderRetracted, EComparisonType.equals, EDataType.binary, TRUE, 0, '', TRUE);
	m_precondition: BoolExpression(m_compExpr65, EBoolOperation.and_op, m_compExpr67);
	
	// (EProcessVariables.Crane_HoldingWorkpiece = FALSE) AND (EProcessVariables.Crane_CylinderRetracted = TRUE)
	m_compExpr70: ComparisonExpression(EProcessVariables.Crane_HoldingWorkpiece, EComparisonType.equals, EDataType.binary, FALSE, 0, '', TRUE);
	m_compExpr72: ComparisonExpression(EProcessVariables.Crane_CylinderRetracted, EComparisonType.equals, EDataType.binary, TRUE, 0, '', TRUE);
	m_postcondition: BoolExpression(m_compExpr70, EBoolOperation.and_op, m_compExpr72);
END_VAR

SUPER^();

METHOD Abort : BOOL
VAR_INPUT
END_VAR
m_ptrCrane^.o_MonostableCylinder.METH_Retract();
IF m_ptrCrane^.o_VacuumGripper.WPTaken THEN
	m_ptrCrane^.o_VacuumGripper.METH_Intake();
ELSE
	m_ptrCrane^.o_VacuumGripper.METH_Release();
END_IF
Abort := TRUE;
END_METHOD

(* Execution logic of this Control Primitive. *)
METHOD PROTECTED  ExecuteInternal : BOOL
VAR_INPUT
	i_params: ParameterSet;
END_VAR
CASE m_step OF

	0:	// extend
		m_ptrCrane^.o_MonostableCylinder.METH_Extend();
		IF m_ptrCrane^.o_MonostableCylinder.Extended THEN
			m_step := 1;
		END_IF
	
	1:	// release
		m_ptrCrane^.o_VacuumGripper.METH_Release();
		m_timer(IN := TRUE, PT := T#100MS);
		IF m_timer.Q THEN
			m_timer(IN := FALSE);
			m_step := 2;
		END_IF
		
	2: // shift register
		IF ShiftProduct(FALSE) THEN
			m_step := 3;
		END_IF
	
	3:	// retract
		m_ptrCrane^.o_MonostableCylinder.METH_Retract();
		IF m_ptrCrane^.o_MonostableCylinder.Retracted THEN
			m_step := 0;
			ExecuteInternal := TRUE;
		END_IF	
END_CASE
END_METHOD

METHOD FB_init : BOOL
VAR_INPUT
	bInitRetains : BOOL; // if TRUE, the retain variables are initialized (warm start / cold start)
	bInCopyCode : BOOL;  // if TRUE, the instance afterwards gets moved into the copy code (online change)
	
	i_ptrCrane: POINTER TO Crane;
END_VAR
m_ptrCrane := i_ptrCrane;

m_id := EPrimitives.Crane_PutDownWP;
m_timeout := T#20S;

Precondition := m_precondition;
Postcondition := m_postcondition;
END_METHOD

END_FUNCTION_BLOCK

// ---- 03_ControlPrimitives/Carrier/PickAlpha/PicAlpha_MoveBase.TcPOU
FUNCTION_BLOCK PicAlpha_MoveBase EXTENDS ControlPrimitiveBase
VAR_INPUT
END_VAR
VAR_OUTPUT
END_VAR
VAR
	m_ptrPicAlpha: POINTER TO PicAlpha;
	
	m_initDirection: BOOL; //TRUE: towards Pos4, FALSE: towards Pos1
	m_step: INT := 0;
	
	m_targettimer: TON;
	m_targetTimeout: TIME;
END_VAR

SUPER^();

METHOD Abort : BOOL
VAR_INPUT
END_VAR
m_ptrPicAlpha^.METH_CarrierStop();
Abort := TRUE;
END_METHOD

METHOD AtTarget : BOOL
VAR_INPUT
END_VAR
END_METHOD

(* Execution logic of this Control Primitive. *)
METHOD PROTECTED  ExecuteInternal : BOOL
VAR_INPUT
	i_params: ParameterSet;
END_VAR
CASE m_step OF 
	0: 
		m_targettimer(IN := TRUE, PT := m_targetTimeout);
		IF AtTarget() THEN
			m_step := 2;
			m_targettimer(IN:= FALSE);
		ELSIF m_targettimer.Q THEN
			m_step := 1;
			m_targettimer(IN:= FALSE);
			m_initDirection := NOT m_initDirection;
		END_IF
		
		IF m_initDirection THEN
			m_ptrPicAlpha^.METH_CarrierForward();
		ELSIF NOT m_initDirection THEN
			m_ptrPicAlpha^.METH_CarrierBackward();
		END_IF
		
	1:
		IF AtTarget() THEN
			m_step := 2;
			m_initDirection := NOT m_initDirection;
		END_IF
		IF m_initDirection THEN
			m_ptrPicAlpha^.METH_CarrierForward();
		ELSIF NOT m_initDirection THEN
			m_ptrPicAlpha^.METH_CarrierBackward();
		END_IF
		
	2:
		m_ptrPicAlpha^.METH_CarrierStop();
		ExecuteInternal := TRUE;
		m_step := 0;
	
END_CASE
END_METHOD

END_FUNCTION_BLOCK

// ---- 05_HardwareControl/EquipmentModule/Carriers/PicAlpha.TcPOU
FUNCTION_BLOCK PicAlpha EXTENDS BaseCarrier
VAR_INPUT
END_VAR
VAR_OUTPUT
	o_VacuumGripper: VacuumGripper;
	o_MonostableCylinder: MonostableCylinder;
	o_Distance: INT := 50;
END_VAR
VAR
	m_PresenceSensorPosition1: PresenceSensor;
	m_PresenceSensorPosition2: PresenceSensor;
	m_PresenceSensorPosition3: PresenceSensor;
	m_PresenceSensorPosition4: PresenceSensor;

END_VAR

METHOD METH_CarrierBackward : BOOL
VAR_INPUT
END_VAR
Motor.ACT_TurnCounterclockwise();

IF m_PresenceSensorPosition1.Value THEN
	o_Distance := 0;
ELSIF m_PresenceSensorPosition2.Value THEN
	o_Distance := 10;
ELSIF m_PresenceSensorPosition3.Value THEN
	o_Distance := 50;
ELSIF m_PresenceSensorPosition4.Value THEN
	o_Distance := 100;
END_IF
END_METHOD

METHOD METH_CarrierForward : BOOL
VAR_INPUT
END_VAR
Motor.ACT_TurnClockwise();

IF m_PresenceSensorPosition1.Value THEN
	o_Distance := 0;
ELSIF m_PresenceSensorPosition2.Value THEN
	o_Distance := 10;
ELSIF m_PresenceSensorPosition3.Value THEN
	o_Distance := 50;
ELSIF m_PresenceSensorPosition4.Value THEN
	o_Distance := 100;
END_IF
END_METHOD

METHOD METH_CarrierStop : BOOL
VAR_INPUT
END_VAR
Motor.ACT_Stop();
END_METHOD

PROPERTY PresenceSensorPosition1Value : BOOL
GET
PresenceSensorPosition1Value := m_PresenceSensorPosition1.Value;
END_GET
END_PROPERTY

PROPERTY PresenceSensorPosition2Value : BOOL
GET
PresenceSensorPosition2Value := m_PresenceSensorPosition2.Value;
END_GET
END_PROPERTY

PROPERTY PresenceSensorPosition3Value : BOOL
GET
PresenceSensorPosition3Value := m_PresenceSensorPosition3.Value;
END_GET
END_PROPERTY

PROPERTY PresenceSensorPosition4Value : BOOL
GET
PresenceSensorPosition4Value := m_PresenceSensorPosition4.Value;
END_GET
END_PROPERTY

END_FUNCTION_BLOCK

// ---- 03_ControlPrimitives/Carrier/PickAlpha/PicAlpha_MoveToPos1.TcPOU
FUNCTION_BLOCK PicAlpha_MoveToPos1 EXTENDS PicAlpha_MoveBase
VAR_INPUT
END_VAR
VAR_OUTPUT
END_VAR
VAR
	// EProcessVariables.PicAlpha_CylinderRetracted = TRUE
	m_precondition: ComparisonExpression(EProcessVariables.PicAlpha_CylinderRetracted, EComparisonType.equals, EDataType.binary, TRUE, 0, '', TRUE);
	
	// (EProcessVariables.PicAlpha_AtPos1 = TRUE) AND (EProcessVariables.PicAlpha_CylinderRetracted = TRUE)
	m_compExpr157: ComparisonExpression(EProcessVariables.PicAlpha_AtPos1, EComparisonType.equals, EDataType.binary, TRUE, 0, '', TRUE);
	m_compExpr159: ComparisonExpression(EProcessVariables.PicAlpha_CylinderRetracted, EComparisonType.equals, EDataType.binary, TRUE, 0, '', TRUE);
	m_postcondition: BoolExpression(m_compExpr157, EBoolOperation.and_op, m_compExpr159);
	END_VAR

SUPER^();

METHOD AtTarget : BOOL
VAR_INPUT
END_VAR
AtTarget := m_ptrPicAlpha^.PresenceSensorPosition1Value AND NOT (m_ptrPicAlpha^.PresenceSensorPosition3Value OR m_ptrPicAlpha^.PresenceSensorPosition4Value);
END_METHOD

METHOD FB_init : BOOL
VAR_INPUT
	bInitRetains : BOOL; // if TRUE, the retain variables are initialized (warm start / cold start)
	bInCopyCode : BOOL;  // if TRUE, the instance afterwards gets moved into the copy code (online change)
	
	i_ptrPicAlpha : POINTER TO PicAlpha;
END_VAR
m_ptrPicAlpha := i_ptrPicAlpha;

m_id := EPrimitives.PicAlpha_MoveToPos1;
m_timeout := T#20S;

Precondition := m_precondition;
Postcondition := m_postcondition;

m_initDirection := FALSE;	//TRUE: towards Pos1
m_targetTimeout := T#10S;
END_METHOD

END_FUNCTION_BLOCK

// ---- 03_ControlPrimitives/Carrier/PickAlpha/PicAlpha_MoveToPos2.TcPOU
FUNCTION_BLOCK PicAlpha_MoveToPos2 EXTENDS PicAlpha_MoveBase
VAR_INPUT
END_VAR
VAR_OUTPUT
END_VAR
VAR
	// EProcessVariables.PicAlpha_CylinderRetracted = TRUE
	m_precondition: ComparisonExpression(EProcessVariables.PicAlpha_CylinderRetracted, EComparisonType.equals, EDataType.binary, TRUE, 0, '', TRUE);
	
	// (EProcessVariables.PicAlpha_AtPos2 = TRUE) AND (EProcessVariables.PicAlpha_CylinderRetracted = TRUE)
	m_compExpr164: ComparisonExpression(EProcessVariables.PicAlpha_AtPos2, EComparisonType.equals, EDataType.binary, TRUE, 0, '', TRUE);
	m_compExpr166: ComparisonExpression(EProcessVariables.PicAlpha_CylinderRetracted, EComparisonType.equals, EDataType.binary, TRUE, 0, '', TRUE);
	m_postcondition: BoolExpression(m_compExpr164, EBoolOperation.and_op, m_compExpr166);
END_VAR

SUPER^();

METHOD AtTarget : BOOL
VAR_INPUT
END_VAR
AtTarget := m_ptrPicAlpha^.PresenceSensorPosition2Value AND NOT (m_ptrPicAlpha^.PresenceSensorPosition3Value OR m_ptrPicAlpha^.PresenceSensorPosition4Value);
END_METHOD

METHOD FB_init : BOOL
VAR_INPUT
	bInitRetains : BOOL; // if TRUE, the retain variables are initialized (warm start / cold start)
	bInCopyCode : BOOL;  // if TRUE, the instance afterwards gets moved into the copy code (online change)
	
	i_ptrPicAlpha : POINTER TO PicAlpha;
END_VAR
m_ptrPicAlpha := i_ptrPicAlpha;

m_id := EPrimitives.PicAlpha_MoveToPos2;
m_timeout := T#20S;

Precondition := m_precondition;
Postcondition := m_postcondition;

m_initDirection := FALSE;	//TRUE: towards Pos1
m_targetTimeout := T#10S;
END_METHOD

END_FUNCTION_BLOCK

// ---- 03_ControlPrimitives/Carrier/PickAlpha/PicAlpha_MoveToPos3.TcPOU
FUNCTION_BLOCK PicAlpha_MoveToPos3 EXTENDS PicAlpha_MoveBase
VAR_INPUT
END_VAR
VAR_OUTPUT
END_VAR
VAR
	// EProcessVariables.PicAlpha_CylinderRetracted = TRUE
	m_precondition: ComparisonExpression(EProcessVariables.PicAlpha_CylinderRetracted, EComparisonType.equals, EDataType.binary, TRUE, 0, '', TRUE);
	
	// (EProcessVariables.PicAlpha_AtPos3 = TRUE) AND (EProcessVariables.PicAlpha_CylinderRetracted = TRUE)
	m_compExpr171: ComparisonExpression(EProcessVariables.PicAlpha_AtPos3, EComparisonType.equals, EDataType.binary, TRUE, 0, '', TRUE);
	m_compExpr173: ComparisonExpression(EProcessVariables.PicAlpha_CylinderRetracted, EComparisonType.equals, EDataType.binary, TRUE, 0, '', TRUE);
	m_postcondition: BoolExpression(m_compExpr171, EBoolOperation.and_op, m_compExpr173);
END_VAR

SUPER^();

METHOD AtTarget : BOOL
VAR_INPUT
END_VAR
AtTarget := m_ptrPicAlpha^.PresenceSensorPosition3Value AND NOT (m_ptrPicAlpha^.PresenceSensorPosition1Value OR m_ptrPicAlpha^.PresenceSensorPosition2Value OR m_ptrPicAlpha^.PresenceSensorPosition4Value);
END_METHOD

METHOD FB_init : BOOL
VAR_INPUT
	bInitRetains : BOOL; // if TRUE, the retain variables are initialized (warm start / cold start)
	bInCopyCode : BOOL;  // if TRUE, the instance afterwards gets moved into the copy code (online change)
	
	i_ptrPicAlpha : POINTER TO PicAlpha;
END_VAR
m_ptrPicAlpha := i_ptrPicAlpha;

m_id := EPrimitives.PicAlpha_MoveToPos3;
m_timeout := T#20S;

Precondition := m_precondition;
Postcondition := m_postcondition;

m_initDirection := TRUE;	//TRUE: towards Pos4
m_targetTimeout := T#10S;
END_METHOD

END_FUNCTION_BLOCK

// ---- 03_ControlPrimitives/Carrier/PickAlpha/PicAlpha_MoveToPos4.TcPOU
FUNCTION_BLOCK PicAlpha_MoveToPos4 EXTENDS PicAlpha_MoveBase
VAR_INPUT
END_VAR
VAR_OUTPUT
END_VAR
VAR
	// EProcessVariables.PicAlpha_CylinderRetracted = TRUE
	m_precondition: ComparisonExpression(EProcessVariables.PicAlpha_CylinderRetracted, EComparisonType.equals, EDataType.binary, TRUE, 0, '', TRUE);
	
	// (EProcessVariables.PicAlpha_AtPos4 = TRUE) AND ((EProcessVariables.PicAlpha_CylinderRetracted = TRUE) AND ((EProcessVariables.SSC_ProductType_1 = 0) AND (EProcessVariables.SSC_ProductType_2 = 0)))
	m_compExpr178: ComparisonExpression(EProcessVariables.PicAlpha_AtPos4, EComparisonType.equals, EDataType.binary, TRUE, 0, '', TRUE);
	m_compExpr180: ComparisonExpression(EProcessVariables.PicAlpha_CylinderRetracted, EComparisonType.equals, EDataType.binary, TRUE, 0, '', TRUE);
	m_compExpr182: ComparisonExpression(EProcessVariables.SSC_ProductType_1, EComparisonType.equals, EDataType.numeric, FALSE, 0, '', TRUE);
	m_compExpr184: ComparisonExpression(EProcessVariables.SSC_ProductType_2, EComparisonType.equals, EDataType.numeric, FALSE, 0, '', TRUE);
	m_boolExpr185: BoolExpression(m_compExpr182, EBoolOperation.and_op, m_compExpr184);
	m_boolExpr186: BoolExpression(m_compExpr180, EBoolOperation.and_op, m_boolExpr185);
	m_postcondition: BoolExpression(m_compExpr178, EBoolOperation.and_op, m_boolExpr186);
END_VAR

SUPER^();

METHOD AtTarget : BOOL
VAR_INPUT
END_VAR
AtTarget := m_ptrPicAlpha^.PresenceSensorPosition4Value AND NOT (m_ptrPicAlpha^.PresenceSensorPosition1Value OR m_ptrPicAlpha^.PresenceSensorPosition2Value OR m_ptrPicAlpha^.PresenceSensorPosition3Value);
END_METHOD

METHOD FB_init : BOOL
VAR_INPUT
	bInitRetains : BOOL; // if TRUE, the retain variables are initialized (warm start / cold start)
	bInCopyCode : BOOL;  // if TRUE, the instance afterwards gets moved into the copy code (online change)
	
	i_ptrPicAlpha : POINTER TO PicAlpha;
END_VAR
m_ptrPicAlpha := i_ptrPicAlpha;

m_id := EPrimitives.PicAlpha_MoveToPos4;
m_timeout := T#20S;

Precondition := m_precondition;
Postcondition := m_postcondition;

m_initDirection := TRUE;	//TRUE: towards Pos4
m_targetTimeout := T#10S;
END_METHOD

END_FUNCTION_BLOCK

// ---- 03_ControlPrimitives/Carrier/PickAlpha/PicAlpha_PickUpWP.TcPOU
FUNCTION_BLOCK PicAlpha_PickUpWP EXTENDS ControlPrimitiveBase
VAR_INPUT
END_VAR
VAR_OUTPUT
END_VAR
VAR
	m_ptrPicAlpha: POINTER TO PicAlpha;
	
	m_step: INT := 0;
	m_timer: TON;
	
	// (EProcessVariables.PicAlpha_CylinderRetracted = TRUE) AND (EProcessVariables.PicAlpha_HoldingWorkpiece = FALSE)
	m_compExpr189: ComparisonExpression(EProcessVariables.PicAlpha_CylinderRetracted, EComparisonType.equals, EDataType.binary, TRUE, 0, '', TRUE);
	m_compExpr191: ComparisonExpression(EProcessVariables.PicAlpha_HoldingWorkpiece, EComparisonType.equals, EDataType.binary, FALSE, 0, '', TRUE);
	m_precondition: BoolExpression(m_compExpr189, EBoolOperation.and_op, m_compExpr191);
	
	// (EProcessVariables.PicAlpha_CylinderRetracted = TRUE) AND (EProcessVariables.PicAlpha_HoldingWorkpiece = TRUE)
	m_compExpr194: ComparisonExpression(EProcessVariables.PicAlpha_CylinderRetracted, EComparisonType.equals, EDataType.binary, TRUE, 0, '', TRUE);
	m_compExpr196: ComparisonExpression(EProcessVariables.PicAlpha_HoldingWorkpiece, EComparisonType.equals, EDataType.binary, TRUE, 0, '', TRUE);
	m_postcondition: BoolExpression(m_compExpr194, EBoolOperation.and_op, m_compExpr196);
END_VAR

SUPER^();

METHOD Abort : BOOL
VAR_INPUT
END_VAR
m_ptrPicAlpha^.o_MonostableCylinder.METH_Retract();
IF m_ptrPicAlpha^.o_VacuumGripper.WPTaken THEN
	m_ptrPicAlpha^.o_VacuumGripper.METH_Intake();
ELSE
	m_ptrPicAlpha^.o_VacuumGripper.METH_Release();
END_IF
Abort := TRUE;
END_METHOD

(* Execution logic of this Control Primitive. *)
METHOD PROTECTED  ExecuteInternal : BOOL
VAR_INPUT
	i_params: ParameterSet;
END_VAR
CASE m_step OF

	0:	// extend
		m_ptrPicAlpha^.o_MonostableCylinder.METH_Extend();
		IF m_ptrPicAlpha^.o_MonostableCylinder.Extended THEN
			m_step := 1;
		END_IF
	
	1:	// grip
		m_ptrPicAlpha^.o_VacuumGripper.METH_Intake();
		m_timer(IN := TRUE, PT := T#200MS);
		IF m_timer.Q THEN
			m_timer(IN := FALSE);
			m_step := 2;
		END_IF
	
	2:	// retract
		m_ptrPicAlpha^.o_MonostableCylinder.METH_Retract();
		IF m_ptrPicAlpha^.o_MonostableCylinder.Retracted THEN
			m_step := 0;
			ExecuteInternal := TRUE;
		END_IF	
END_CASE
END_METHOD

METHOD FB_init : BOOL
VAR_INPUT
	bInitRetains : BOOL; // if TRUE, the retain variables are initialized (warm start / cold start)
	bInCopyCode : BOOL;  // if TRUE, the instance afterwards gets moved into the copy code (online change)
	
	i_ptrPicAlpha : POINTER TO PicAlpha;
END_VAR
m_ptrPicAlpha := i_ptrPicAlpha;

m_id := EPrimitives.PicAlpha_PickUpWp;
m_timeout := T#20S;

Precondition := m_precondition;
Postcondition := m_postcondition;
END_METHOD

END_FUNCTION_BLOCK

// ---- 03_ControlPrimitives/Carrier/PickAlpha/PicAlpha_PutDownWP.TcPOU
FUNCTION_BLOCK PicAlpha_PutDownWP EXTENDS ControlPrimitiveBase
VAR_INPUT
END_VAR
VAR_OUTPUT
END_VAR
VAR
	m_ptrPicAlpha: POINTER TO PicAlpha;
	m_ptrPAC: POINTER TO PicAlphaConveyor;
	
	m_step: INT := 0;
	m_timer: TON;
	
	// (EProcessVariables.PicAlpha_CylinderRetracted = TRUE) AND (EProcessVariables.PicAlpha_HoldingWorkpiece = TRUE)
	m_compExpr199: ComparisonExpression(EProcessVariables.PicAlpha_CylinderRetracted, EComparisonType.equals, EDataType.binary, TRUE, 0, '', TRUE);
	m_compExpr201: ComparisonExpression(EProcessVariables.PicAlpha_HoldingWorkpiece, EComparisonType.equals, EDataType.binary, TRUE, 0, '', TRUE);
	m_precondition: BoolExpression(m_compExpr199, EBoolOperation.and_op, m_compExpr201);
	
	// (EProcessVariables.PicAlpha_CylinderRetracted = TRUE) AND (EProcessVariables.PicAlpha_HoldingWorkpiece = FALSE)
	m_compExpr204: ComparisonExpression(EProcessVariables.PicAlpha_CylinderRetracted, EComparisonType.equals, EDataType.binary, TRUE, 0, '', TRUE);
	m_compExpr206: ComparisonExpression(EProcessVariables.PicAlpha_HoldingWorkpiece, EComparisonType.equals, EDataType.binary, FALSE, 0, '', TRUE);
	m_postcondition: BoolExpression(m_compExpr204, EBoolOperation.and_op, m_compExpr206);
END_VAR

SUPER^();

METHOD Abort : BOOL
VAR_INPUT
END_VAR
m_ptrPicAlpha^.o_MonostableCylinder.METH_Retract();
IF m_ptrPicAlpha^.o_VacuumGripper.WPTaken THEN
	m_ptrPicAlpha^.o_VacuumGripper.METH_Intake();
ELSE
	m_ptrPicAlpha^.o_VacuumGripper.METH_Release();
END_IF
Abort := TRUE;
END_METHOD

(* Execution logic of this Control Primitive. *)
METHOD PROTECTED  ExecuteInternal : BOOL
VAR_INPUT
	i_params: ParameterSet;
END_VAR
CASE m_step OF

	0:	// extend
		m_ptrPicAlpha^.o_MonostableCylinder.METH_Extend();
		IF m_ptrPicAlpha^.o_MonostableCylinder.Extended THEN
			m_step := 1;
		END_IF
	
	1:	// grip
		m_ptrPicAlpha^.o_VacuumGripper.METH_Release();
		m_ptrPicAlpha^.o_VacuumGripper.METH_VacuumHitOn();
		m_timer(IN := TRUE, PT := T#200MS);
		IF m_timer.Q THEN
			m_ptrPicAlpha^.o_VacuumGripper.METH_VacuumHitOff();
			m_timer(IN := FALSE);
			m_step := 2;
			IF m_ptrPicAlpha^.PresenceSensorPosition4Value THEN
				m_ptrPAC^.METH_ReduceWPNumberAtPAC();
			END_IF
		END_IF
	
	2:	// retract
		m_ptrPicAlpha^.o_MonostableCylinder.METH_Retract();
		IF m_ptrPicAlpha^.o_MonostableCylinder.Retracted THEN
			m_step := 0;
			ExecuteInternal := TRUE;
		END_IF	
END_CASE
END_METHOD

METHOD FB_init : BOOL
VAR_INPUT
	bInitRetains : BOOL; // if TRUE, the retain variables are initialized (warm start / cold start)
	bInCopyCode : BOOL;  // if TRUE, the instance afterwards gets moved into the copy code (online change)
	
	i_ptrPicAlpha : POINTER TO PicAlpha;
	i_ptrPAC : POINTER TO PicAlphaConveyor;
END_VAR
m_ptrPicAlpha := i_ptrPicAlpha;
m_ptrPAC := i_ptrPAC;

m_id := EPrimitives.PicAlpha_PutDownWp;
m_timeout := T#20S;

Precondition := m_precondition;
Postcondition := m_postcondition;
END_METHOD

END_FUNCTION_BLOCK

// ---- 05_HardwareControl/EquipmentModule/Conveyors/PicAlphaConveyor.TcPOU
FUNCTION_BLOCK PicAlphaConveyor EXTENDS Conveyor
VAR_INPUT
END_VAR
VAR_OUTPUT
END_VAR
VAR
	//Sensors
	m_PresencesensorStart : PresenceSensor;
	m_PresencesensorEnd : PresenceSensor;
	
	m_Switch: Switch;
	m_WPNumberAtPAC : INT := 0;
END_VAR

METHOD METH_IncreaseWPNumberAtPAC : BOOL
VAR_INPUT
END_VAR
m_WPNumberAtPAC := m_WPNumberAtPAC + 1;
END_METHOD

METHOD METH_ReduceWPNumberAtPAC : BOOL
VAR_INPUT
END_VAR
m_WPNumberAtPAC := m_WPNumberAtPAC - 1;
END_METHOD

METHOD METH_ResetWPNumberAtPAC : BOOL
VAR_INPUT
END_VAR
m_WPNumberAtPAC := 0;
END_METHOD

METHOD METH_Switch_Extend : BOOL
VAR_INPUT
END_VAR
m_Switch.METH_Extend();
END_METHOD

METHOD METH_Switch_Retract : BOOL
VAR_INPUT
END_VAR
m_Switch.METH_Retract();
END_METHOD

PROPERTY WPAtEnd : BOOL
GET
WPAtEnd := m_presenceSensorEnd.Value;
END_GET
END_PROPERTY

PROPERTY WPAtStart : BOOL
GET
WPAtStart := m_presenceSensorStart.Value;
END_GET
END_PROPERTY

END_FUNCTION_BLOCK

// ---- 05_HardwareControl/EquipmentModule/Conveyors/Conveyor.TcPOU
FUNCTION_BLOCK Conveyor EXTENDS BaseComponent
VAR_INPUT
END_VAR
VAR_OUTPUT
END_VAR
VAR
	Motor : Motor;
END_VAR

METHOD METH_ConveyorBackward : BOOL
VAR_INPUT
END_VAR
Motor.ACT_TurnCounterclockwise();
END_METHOD

METHOD METH_ConveyorForward : BOOL
VAR_INPUT
END_VAR
Motor.ACT_TurnClockwise();
END_METHOD

METHOD METH_ConveyorStop : BOOL
VAR_INPUT
END_VAR
Motor.ACT_Stop();
END_METHOD

END_FUNCTION_BLOCK

// ---- 05_HardwareControl/ControlModule/Pushers/Switch.TcPOU
FUNCTION_BLOCK Switch IMPLEMENTS ITF_Cylinder
VAR_INPUT
END_VAR
VAR_OUTPUT
END_VAR
VAR
	//Hardware
	DI_Extended AT %I* : BOOL;
	DI_Retracted AT %I* : BOOL;
	DO_Extend AT %Q* : BOOL;
	//NOT USED BUT USABLE
	DI_BoundaryPressure AT %I* : BOOL;
END_VAR

PROPERTY Extended : BOOL
GET
Extended := DI_Extended;
END_GET
END_PROPERTY

METHOD METH_Extend : BOOL
DO_Extend := TRUE;
END_METHOD

METHOD METH_Retract : BOOL
DO_Extend := FALSE;
END_METHOD

PROPERTY Retracted : BOOL
GET
Retracted := DI_Retracted;
END_GET
END_PROPERTY

END_FUNCTION_BLOCK

// ---- 03_ControlPrimitives/Conveyor/LSC/LSC_MoveWorkpiece_Base.TcPOU
FUNCTION_BLOCK ABSTRACT LSC_MoveWorkpiece_Base EXTENDS ControlPrimitiveBase
VAR_INPUT
END_VAR
VAR_OUTPUT
END_VAR
VAR
	m_ptrLSC: POINTER TO LargeSortingConveyor;
	
	m_step: INT := 0;
END_VAR

SUPER^();

METHOD Abort : BOOL
VAR_INPUT
END_VAR
m_ptrLSC^.METH_ConveyorStop();
m_ptrLSC^.METH_Ramp1Pusher_Retract();
m_ptrLSC^.METH_Ramp2Pusher_Retract();
m_ptrLSC^.METH_Switch_Retract();
Abort := TRUE;
END_METHOD

METHOD PROTECTED ABSTRACT AtTarget : BOOL
VAR_INPUT
END_VAR
END_METHOD

METHOD PROTECTED ABSTRACT EjectOperation : BOOL
VAR_INPUT
END_VAR
END_METHOD

(* Execution logic of this Control Primitive. *)
METHOD PROTECTED ExecuteInternal : BOOL
VAR_INPUT
	i_params: ParameterSet;
END_VAR
CASE m_step OF
	0: // to target	
	IF NOT AtTarget() THEN
		m_ptrLSC^.METH_ConveyorForward();
		m_step := 1;
	END_IF
	
	1:
	IF AtTarget() THEN
		m_ptrLSC^.METH_ConveyorStop();
		m_ptrLSC^.METH_Switch_Retract();
		m_step := 2;
	END_IF
	
	2:
	IF EjectOperation() THEN
		m_step := 0;
		ExecuteInternal := TRUE;
	END_IF
		
END_CASE
END_METHOD

END_FUNCTION_BLOCK

// ---- 05_HardwareControl/EquipmentModule/Conveyors/LargeSortingConveyor.TcPOU
FUNCTION_BLOCK LargeSortingConveyor EXTENDS Conveyor
VAR_INPUT
END_VAR
VAR_OUTPUT
END_VAR
VAR
	m_rampPusherStart : MonostableCylinder;
	m_rampPusherMid : MonostableCylinder;
	m_Switch : Switch;
	
	m_presenceSensorStart : PresenceSensor;
	m_opticalSensorStart : OpticalSensor;
	m_opticalSensorMid : OpticalSensor;
	m_opticalSensorEnd : OpticalSensor;
	m_inductiveSensorStart : InductiveSensor;
	m_inductiveSensorMid : InductiveSensor;
	
	m_rampStart : Ramp;
	m_rampMiddle : Ramp;
	m_rampEnd : Ramp;
END_VAR

PROPERTY LightWPAtEnd : BOOL
GET
LightWPAtEnd := m_opticalSensorEnd.Value;
END_GET
END_PROPERTY

PROPERTY LightWPAtMid : BOOL
GET
LightWPAtMid := m_opticalSensorMid.Value;
END_GET
END_PROPERTY

PROPERTY LightWPAtStart : BOOL
GET
LightWPAtStart := m_opticalSensorStart.Value;
END_GET
END_PROPERTY

PROPERTY MetalWPAtMid : BOOL
GET
MetalWPAtMid := m_inductiveSensorMid.Value;
END_GET
END_PROPERTY

PROPERTY MetalWPAtStart : BOOL
GET
MetalWPAtStart := m_inductiveSensorStart.Value;
END_GET
END_PROPERTY

METHOD METH_Ramp1Pusher_Extend : BOOL
VAR_INPUT
END_VAR
m_rampPusherStart.METH_Extend();
END_METHOD

METHOD METH_Ramp1Pusher_Retract : BOOL
VAR_INPUT
END_VAR
m_rampPusherStart.METH_Retract();
END_METHOD

METHOD METH_Ramp2Pusher_Extend : BOOL
VAR_INPUT
END_VAR
m_rampPusherMid.METH_Extend();
END_METHOD

METHOD METH_Ramp2Pusher_Retract : BOOL
VAR_INPUT
END_VAR
m_rampPusherMid.METH_Retract();
END_METHOD

METHOD METH_Switch_Extend : BOOL
VAR_INPUT
END_VAR
m_Switch.METH_Extend();
END_METHOD

METHOD METH_Switch_Retract : BOOL
VAR_INPUT
END_VAR
m_Switch.METH_Retract();
END_METHOD

PROPERTY WPAtRampEnd : BOOL
GET
WPAtRampEnd := m_rampEnd.m_presenceSensorRampFull.Value;
END_GET
END_PROPERTY

PROPERTY WPAtRampMiddle : BOOL
GET
WPAtRampMiddle := m_rampMiddle.m_presenceSensorRampFull.Value;
END_GET
END_PROPERTY

PROPERTY WPAtRampStart : BOOL
GET
WPAtRampStart := m_rampStart.m_presenceSensorRampFull.Value;
END_GET
END_PROPERTY

PROPERTY WPAtStart : BOOL
GET
WPAtStart := m_presenceSensorStart.Value;
END_GET
END_PROPERTY

END_FUNCTION_BLOCK

// ---- 05_HardwareControl/ControlModule/Sensors/OpticalSensor.TcPOU
FUNCTION_BLOCK OpticalSensor IMPLEMENTS ITF_BinarySensor
VAR_INPUT
END_VAR
VAR_OUTPUT
END_VAR
VAR
	//Hardware
	DI_WPLight AT %I* : BOOL;
END_VAR

PROPERTY Value : BOOL
GET
Value := DI_WPLight;
END_GET
END_PROPERTY

END_FUNCTION_BLOCK

// ---- 05_HardwareControl/ControlModule/Sensors/InductiveSensor.TcPOU
FUNCTION_BLOCK InductiveSensor IMPLEMENTS ITF_BinarySensor
VAR_INPUT
END_VAR
VAR_OUTPUT
END_VAR
VAR
	//Hardware
	DI_WPMetallic AT %I* : BOOL;
END_VAR

PROPERTY Value : BOOL
GET
Value := DI_WPMetallic;
END_GET
END_PROPERTY

END_FUNCTION_BLOCK

// ---- 05_HardwareControl/EquipmentModule/Ramps/Ramp.TcPOU
FUNCTION_BLOCK Ramp
VAR_INPUT
END_VAR
VAR_OUTPUT
	m_presenceSensorRampFull : PresenceSensor;
END_VAR
VAR
END_VAR

END_FUNCTION_BLOCK

// ---- 03_ControlPrimitives/Conveyor/LSC/LSC_SearchWorkpiece.TcPOU
FUNCTION_BLOCK LSC_SearchWorkpiece EXTENDS ControlPrimitiveBase
VAR_INPUT
END_VAR
VAR_OUTPUT
END_VAR
VAR
	m_ptrLSC: POINTER TO LargeSortingConveyor;
	
	// TRUE
	m_precondition: ValueExpression(EDataType.binary, TRUE, 0, '', TRUE);
	
	// EProcessVariables.LSC_ProductType >= 0
	m_postcondition: ComparisonExpression(EProcessVariables.LSC_ProductType, EComparisonType.greater_eq, EDataType.numeric, FALSE, 0, '', TRUE);
	
	m_timer: TON;
	m_passby: BOOL;
	m_step: INT := 0;
END_VAR

SUPER^();

METHOD Abort : BOOL
VAR_INPUT
END_VAR
m_ptrLSC^.METH_ConveyorStop();
m_ptrLSC^.METH_Ramp1Pusher_Retract();
m_ptrLSC^.METH_Ramp2Pusher_Retract();
m_ptrLSC^.METH_Switch_Retract();
Abort := TRUE;
END_METHOD

(* Execution logic of this Control Primitive. *)
METHOD PROTECTED  ExecuteInternal : BOOL
VAR_INPUT
	i_params: ParameterSet;
END_VAR
//searches for a workpiece on the large sorting conveyor.
//If one is detected it is moved to the identifying sensors. 
//If none is detected, the conveyor is run to move all possible objects of it.

CASE m_step OF
	0:	//search in front of presence sensor
		m_ptrLSC^.METH_ConveyorForward();
		m_timer(IN := TRUE, PT := T#600MS);
		
		IF m_timer.Q THEN	//empty in front of presence sensor
			m_timer(IN := FALSE);
			m_ptrLSC^.METH_ConveyorStop();
			m_step := 1;
		END_IF
		IF m_ptrLSC^.WPAtStart THEN //Workpiece detected
			m_timer(IN := FALSE);
			m_ptrLSC^.METH_ConveyorStop();
			m_step := 2;
		END_IF

	1:	//search behind presence sensor
		m_ptrLSC^.METH_ConveyorBackward();
		m_timer(IN := TRUE, PT := T#3000MS);
		
		IF m_timer.Q THEN	//empty behind presence sensor
			m_timer(IN := FALSE);
			m_ptrLSC^.METH_ConveyorStop();
			m_step := 4;
		END_IF	
		IF m_ptrLSC^.WPAtStart THEN //Workpiece detected
			m_timer(IN := FALSE);			
			m_ptrLSC^.METH_ConveyorStop();
			m_step := 2;
		END_IF

		
	2:	//workpiece found, identify workpiece  (300ms)
		m_ptrLSC^.METH_ConveyorForward();
		m_timer(IN := TRUE, PT := T#300MS);
		
		IF m_timer.Q THEN	//workpiece at inductive and optical sensor
			m_timer(IN := FALSE);
			m_ptrLSC^.METH_ConveyorStop();
			m_step := 3;
		END_IF	

	
	3:	//move workpiece to presence sensor
		m_ptrLSC^.METH_ConveyorBackward();
		IF m_ptrLSC^.WPAtStart THEN
			m_ptrLSC^.METH_ConveyorStop();
			m_step := 0;
			ExecuteInternal := TRUE;
		END_IF
	
		
	4:	//no workpiece found; empty conveyor
		m_ptrLSC^.METH_ConveyorForward();
		m_timer(IN := TRUE, PT := T#4000MS);
		
		IF m_timer.Q THEN	//conveyor is empty 
			m_timer(IN := FALSE);
			m_ptrLSC^.METH_ConveyorStop();
			m_step := 0;
			ExecuteInternal := TRUE;
		END_IF	
	
END_CASE
END_METHOD

METHOD FB_init : BOOL
VAR_INPUT
	bInitRetains : BOOL; // if TRUE, the retain variables are initialized (warm start / cold start)
	bInCopyCode : BOOL;  // if TRUE, the instance afterwards gets moved into the copy code (online change)
	
	i_ptrLSC: POINTER TO LargeSortingConveyor;
END_VAR
m_ptrLSC := i_ptrLSC;

m_id := EPrimitives.LSC_SearchWorkpiece;
m_timeout := T#200S;

Precondition := m_precondition;
Postcondition := m_postcondition;
END_METHOD

END_FUNCTION_BLOCK

// ---- 03_ControlPrimitives/Conveyor/LSC/LSC_TransferWorkpieceTo_PAC.TcPOU
FUNCTION_BLOCK LSC_TransferWorkpieceTo_PAC EXTENDS LSC_MoveWorkpiece_Base
VAR_INPUT
END_VAR
VAR_OUTPUT
END_VAR
VAR
	// (EProcessVariables.PAC_WPNumber < 3) AND (((EProcessVariables.PicAlpha_AtPos1 = FALSE) AND (EProcessVariables.PicAlpha_AtPos2 = FALSE)) OR (EProcessVariables.PicAlpha_CylinderRetracted = TRUE))
	m_compExpr91: ComparisonExpression(EProcessVariables.PAC_WPNumber, EComparisonType.less, EDataType.numeric, FALSE, 3, '', TRUE);
	m_compExpr93: ComparisonExpression(EProcessVariables.PicAlpha_AtPos1, EComparisonType.equals, EDataType.binary, FALSE, 0, '', TRUE);
	m_compExpr95: ComparisonExpression(EProcessVariables.PicAlpha_AtPos2, EComparisonType.equals, EDataType.binary, FALSE, 0, '', TRUE);
	m_boolExpr96: BoolExpression(m_compExpr93, EBoolOperation.and_op, m_compExpr95);
	m_compExpr98: ComparisonExpression(EProcessVariables.PicAlpha_CylinderRetracted, EComparisonType.equals, EDataType.binary, TRUE, 0, '', TRUE);
	m_boolExpr99: BoolExpression(m_boolExpr96, EBoolOperation.or_op, m_compExpr98);
	m_precondition: BoolExpression(m_compExpr91, EBoolOperation.and_op, m_boolExpr99);
	
	// EProcessVariables.PAC_WPAtStart = TRUE
	m_postcondition: ComparisonExpression(EProcessVariables.PAC_WPAtStart, EComparisonType.equals, EDataType.binary, TRUE, 0, '', TRUE);
	
	m_timer: TON;
	m_passby: BOOL;
END_VAR

SUPER^();

METHOD PROTECTED  AtTarget : BOOL
VAR_INPUT
END_VAR
AtTarget := FALSE;
m_ptrLSC^.METH_Switch_Extend();

IF m_ptrLSC^.WPAtStart THEN
	m_passby := TRUE;
END_IF

IF m_passby THEN
	m_timer(IN := TRUE, PT := T#2000MS);
	IF m_timer.Q THEN
		m_timer(IN := FALSE);
		m_passby := FALSE;
		AtTarget := TRUE;
	END_IF
END_IF
END_METHOD

METHOD PROTECTED EjectOperation : BOOL
VAR_INPUT
END_VAR
EjectOperation := FALSE;

m_ptrLSC^.METH_Switch_Extend();
m_ptrLSC^.METH_ConveyorForward();
m_timer(IN := TRUE, PT := T#2S);

IF m_timer.Q THEN
	m_ptrLSC^.METH_Switch_Retract();
	m_ptrLSC^.METH_ConveyorStop();
	m_st^.ShiftProduct(EProducts.LSC_product, EProducts.PAC_product1);
	EjectOperation := TRUE;
END_IF
END_METHOD

METHOD FB_init : BOOL
VAR_INPUT
	bInitRetains : BOOL; // if TRUE, the retain variables are initialized (warm start / cold start)
	bInCopyCode : BOOL;  // if TRUE, the instance afterwards gets moved into the copy code (online change)
	
	i_ptrLSC: POINTER TO LargeSortingConveyor;
END_VAR
m_ptrLSC := i_ptrLSC;

m_id := EPrimitives.LSC_TransferWorkpieceTo_PAC;
m_timeout := T#5S;

Precondition := m_precondition;
Postcondition := m_postcondition;
END_METHOD

END_FUNCTION_BLOCK

// ---- 03_ControlPrimitives/Conveyor/LSC/LSC_TransferWorkpieceTo_RampEnd.TcPOU
FUNCTION_BLOCK LSC_TransferWorkpieceTo_RampEnd EXTENDS LSC_MoveWorkpiece_Base
VAR_INPUT
END_VAR
VAR_OUTPUT
END_VAR
VAR
	// EProcessVariables.LSC_WPAtRampEnd = FALSE
	m_precondition: ComparisonExpression(EProcessVariables.LSC_WPAtRampEnd, EComparisonType.equals, EDataType.binary, FALSE, 0, '', TRUE);
	
	// TRUE
	m_postcondition: ValueExpression(EDataType.binary, TRUE, 0, '', TRUE);
END_VAR

SUPER^();

METHOD PROTECTED  AtTarget : BOOL
VAR_INPUT
END_VAR
AtTarget := m_ptrLSC^.WPAtRampEnd;
END_METHOD

METHOD PROTECTED EjectOperation : BOOL
VAR_INPUT
END_VAR
EjectOperation := TRUE;
m_st^.ShiftProduct(EProducts.LSC_product, 0);
END_METHOD

METHOD FB_init : BOOL
VAR_INPUT
	bInitRetains : BOOL; // if TRUE, the retain variables are initialized (warm start / cold start)
	bInCopyCode : BOOL;  // if TRUE, the instance afterwards gets moved into the copy code (online change)
	
	i_ptrLSC: POINTER TO LargeSortingConveyor;
END_VAR
m_ptrLSC := i_ptrLSC;

m_id := EPrimitives.LSC_TransferWorkpieceTo_RampEnd;
m_timeout := T#200S;

Precondition := m_precondition;
Postcondition := m_postcondition;
END_METHOD

END_FUNCTION_BLOCK

// ---- 03_ControlPrimitives/Conveyor/LSC/LSC_TransferWorkpieceTo_RampMid.TcPOU
FUNCTION_BLOCK LSC_TransferWorkpieceTo_RampMid EXTENDS LSC_MoveWorkpiece_Base
VAR_INPUT
END_VAR
VAR_OUTPUT
END_VAR
VAR
	// EProcessVariables.LSC_WPAtRampMiddle = FALSE
	m_precondition: ComparisonExpression(EProcessVariables.LSC_WPAtRampMiddle, EComparisonType.equals, EDataType.binary, FALSE, 0, '', TRUE);
	
	// TRUE
	m_postcondition: ValueExpression(EDataType.binary, TRUE, 0, '', TRUE);
	
	m_timer: TON;
	m_passby : BOOL;
END_VAR

SUPER^();

METHOD PROTECTED  AtTarget : BOOL
VAR_INPUT
END_VAR
AtTarget := FALSE;

IF m_ptrLSC^.WPAtStart THEN
	m_passby := TRUE;
END_IF

IF m_passby THEN
	m_timer(IN := TRUE, PT := T#2100MS);
	IF m_timer.Q THEN
		m_timer(IN := FALSE);
		m_passby := FALSE;
		AtTarget := TRUE;
	END_IF
END_IF
END_METHOD

METHOD PROTECTED EjectOperation : BOOL
VAR_INPUT
END_VAR
m_ptrLSC^.METH_Ramp2Pusher_Extend();
IF m_ptrLSC^.WPAtRampMiddle THEN
	m_ptrLSC^.METH_Ramp2Pusher_Retract();
	m_st^.ShiftProduct(EProducts.LSC_product, 0);
	EjectOperation := TRUE;
END_IF
END_METHOD

METHOD FB_init : BOOL
VAR_INPUT
	bInitRetains : BOOL; // if TRUE, the retain variables are initialized (warm start / cold start)
	bInCopyCode : BOOL;  // if TRUE, the instance afterwards gets moved into the copy code (online change)
	
	i_ptrLSC: POINTER TO LargeSortingConveyor;
END_VAR
m_ptrLSC := i_ptrLSC;

m_id := EPrimitives.LSC_TransferWorkpieceTo_RampMid;
m_timeout := T#200S;

Precondition := m_precondition;
Postcondition := m_postcondition;
END_METHOD

END_FUNCTION_BLOCK

// ---- 03_ControlPrimitives/Conveyor/LSC/LSC_TransferWorkpieceTo_RampStart.TcPOU
FUNCTION_BLOCK LSC_TransferWorkpieceTo_RampStart EXTENDS LSC_MoveWorkpiece_Base
VAR_INPUT
END_VAR
VAR_OUTPUT
END_VAR
VAR
	// EProcessVariables.LSC_WPAtRampStart = FALSE
	m_precondition: ComparisonExpression(EProcessVariables.LSC_WPAtRampStart, EComparisonType.equals, EDataType.binary, FALSE, 0, '', TRUE);
	
	// TRUE
	m_postcondition: ValueExpression(EDataType.binary, TRUE, 0, '', TRUE);
	
	m_timer: TON;
	m_passby: BOOL;
END_VAR

SUPER^();

METHOD PROTECTED  AtTarget : BOOL
VAR_INPUT
END_VAR
AtTarget := FALSE;

IF m_ptrLSC^.WPAtStart THEN
	m_passby := TRUE;
END_IF

IF m_passby THEN
	m_timer(IN := TRUE, PT := T#700MS);
	IF m_timer.Q THEN
		m_timer(IN := FALSE);
		m_passby := FALSE;
		AtTarget := TRUE;
	END_IF
END_IF
END_METHOD

METHOD PROTECTED EjectOperation : BOOL
VAR_INPUT
END_VAR
m_ptrLSC^.METH_Ramp1Pusher_Extend();
IF m_ptrLSC^.WPAtRampStart THEN
	m_ptrLSC^.METH_Ramp1Pusher_Retract();
	m_st^.ShiftProduct(EProducts.LSC_product, 0);
	EjectOperation := TRUE;
END_IF
END_METHOD

METHOD FB_init : BOOL
VAR_INPUT
	bInitRetains : BOOL; // if TRUE, the retain variables are initialized (warm start / cold start)
	bInCopyCode : BOOL;  // if TRUE, the instance afterwards gets moved into the copy code (online change)
	
	i_ptrLSC: POINTER TO LargeSortingConveyor;
END_VAR
m_ptrLSC := i_ptrLSC;

m_id := EPrimitives.LSC_TransferWorkpieceTo_RampStart;
m_timeout := T#200S;

Precondition := m_precondition;
Postcondition := m_postcondition;
END_METHOD

END_FUNCTION_BLOCK

// ---- 03_ControlPrimitives/Conveyor/PAC/PAC_MoveWorkpiece_Base.TcPOU
FUNCTION_BLOCK ABSTRACT PAC_MoveWorkpiece_Base EXTENDS ControlPrimitiveBase
VAR_INPUT
END_VAR
VAR_OUTPUT
END_VAR
VAR
	m_ptrPAC: POINTER TO PicAlphaConveyor;
	
	m_step: INT := 0;
END_VAR

SUPER^();

METHOD  Abort : BOOL
VAR_INPUT
END_VAR
m_ptrPAC^.METH_ConveyorStop();
m_ptrPAC^.METH_Switch_Retract();
Abort := TRUE;
END_METHOD

METHOD PROTECTED ABSTRACT AtTarget : BOOL
VAR_INPUT
END_VAR
END_METHOD

METHOD PROTECTED ABSTRACT EjectOperation : BOOL
VAR_INPUT
END_VAR
END_METHOD

(* Execution logic of this Control Primitive. *)
METHOD PROTECTED ExecuteInternal : BOOL
VAR_INPUT
	i_params: ParameterSet;
END_VAR
CASE m_step OF
	0: // to target	
	IF NOT AtTarget() THEN
		m_ptrPAC^.METH_ConveyorForward();
		m_step := 1;
	END_IF
		
	1:
	IF AtTarget() THEN
		m_ptrPAC^.METH_ConveyorStop();
		//m_ptrPAC^.METH_Switch_Extend();
		m_step := 2;
	END_IF
	
	2:
	IF EjectOperation() THEN
		m_step := 0;
		ExecuteInternal := TRUE;
	END_IF
		
END_CASE
END_METHOD

END_FUNCTION_BLOCK

// ---- 03_ControlPrimitives/Conveyor/PAC/PAC_TransferWorkpieceTo_PSEnd.TcPOU
FUNCTION_BLOCK PAC_TransferWorkpieceTo_PSEnd EXTENDS PAC_MoveWorkpiece_Base
VAR_INPUT
END_VAR
VAR_OUTPUT
END_VAR
VAR
	// (EProcessVariables.PicAlpha_CylinderRetracted = TRUE) AND (EProcessVariables.PAC_WPAtEnd = FALSE)
	m_compExpr116: ComparisonExpression(EProcessVariables.PicAlpha_CylinderRetracted, EComparisonType.equals, EDataType.binary, TRUE, 0, '', TRUE);
	m_compExpr118: ComparisonExpression(EProcessVariables.PAC_WPAtEnd, EComparisonType.equals, EDataType.binary, FALSE, 0, '', TRUE);
	m_precondition: BoolExpression(m_compExpr116, EBoolOperation.and_op, m_compExpr118);
	
	// EProcessVariables.PAC_WPAtEnd = TRUE
	m_postcondition: ComparisonExpression(EProcessVariables.PAC_WPAtEnd, EComparisonType.equals, EDataType.binary, TRUE, 0, '', TRUE);
	
	m_switchExtended: BOOL;
	m_timer: TON;
END_VAR

SUPER^();

METHOD PROTECTED  AtTarget : BOOL
VAR_INPUT
END_VAR
AtTarget := FALSE;

IF NOT m_switchExtended THEN
	m_ptrPAC^.METH_Switch_Extend();
	m_switchExtended := TRUE;
ELSE
	m_timer(IN := TRUE, PT := T#500MS);
	IF m_timer.Q THEN
		m_ptrPAC^.METH_Switch_Retract();
	END_IF
END_IF

IF m_ptrPAC^.WPAtEnd THEN
	m_timer(IN := FALSE);
	AtTarget := TRUE;
	m_switchExtended := FALSE;
END_IF
END_METHOD

METHOD PROTECTED EjectOperation : BOOL
VAR_INPUT
END_VAR
EjectOperation := TRUE;
END_METHOD

METHOD FB_init : BOOL
VAR_INPUT
	bInitRetains : BOOL; // if TRUE, the retain variables are initialized (warm start / cold start)
	bInCopyCode : BOOL;  // if TRUE, the instance afterwards gets moved into the copy code (online change)
	
	i_ptrPAC: POINTER TO PicAlphaConveyor;
END_VAR
m_ptrPAC := i_ptrPAC;

m_id := EPrimitives.PAC_TransferWorkpieceTo_PSEnd;
m_timeout := T#200S;

Precondition := m_precondition;
Postcondition := m_postcondition;
END_METHOD

END_FUNCTION_BLOCK

// ---- 03_ControlPrimitives/Conveyor/PAC/PAC_TransferWorkpieceTo_PSStart.TcPOU
FUNCTION_BLOCK PAC_TransferWorkpieceTo_PSStart EXTENDS PAC_MoveWorkpiece_Base
VAR_INPUT
END_VAR
VAR_OUTPUT
END_VAR
VAR
	// (EProcessVariables.LSC_ProductType = 4) AND (EProcessVariables.PAC_WPNumber < 3)
	m_compExpr120: ComparisonExpression(EProcessVariables.LSC_ProductType, EComparisonType.equals, EDataType.numeric, FALSE, 4, '', TRUE);
	m_compExpr122: ComparisonExpression(EProcessVariables.PAC_WPNumber, EComparisonType.less, EDataType.numeric, FALSE, 3, '', TRUE);
	m_precondition: BoolExpression(m_compExpr120, EBoolOperation.and_op, m_compExpr122);
	
	// EProcessVariables.PAC_WPAtStart = TRUE
	m_postcondition: ComparisonExpression(EProcessVariables.PAC_WPAtStart, EComparisonType.equals, EDataType.binary, TRUE, 0, '', TRUE);
	
	m_timer: TON;
END_VAR

SUPER^();

METHOD PROTECTED  AtTarget : BOOL
VAR_INPUT
END_VAR
AtTarget := FALSE;

m_timer(IN := TRUE, PT := T#2000MS);
IF m_timer.Q THEN
	m_timer(IN := FALSE);
	m_ptrPAC^.METH_IncreaseWPNumberAtPAC();
	AtTarget := TRUE;
END_IF
END_METHOD

METHOD PROTECTED EjectOperation : BOOL
VAR_INPUT
END_VAR
//m_ptrPAC^.METH_IncreaseWPNumberAtPAC();
EjectOperation := TRUE;
END_METHOD

METHOD FB_init : BOOL
VAR_INPUT
	bInitRetains : BOOL; // if TRUE, the retain variables are initialized (warm start / cold start)
	bInCopyCode : BOOL;  // if TRUE, the instance afterwards gets moved into the copy code (online change)
	
	i_ptrPAC: POINTER TO PicAlphaConveyor;
END_VAR
m_ptrPAC := i_ptrPAC;

m_id := EPrimitives.PAC_TransferWorkpieceTo_PSStart;
m_timeout := T#200S;

Precondition := m_precondition;
Postcondition := m_postcondition;
END_METHOD

END_FUNCTION_BLOCK

// ---- 03_ControlPrimitives/Conveyor/PAC/PAC_TransferWorkpieceTo_SSC.TcPOU
FUNCTION_BLOCK PAC_TransferWorkpieceTo_SSC EXTENDS PAC_MoveWorkpiece_Base
VAR_INPUT
END_VAR
VAR_OUTPUT
END_VAR
VAR
	// (EProcessVariables.PicAlpha_AtPos3 = TRUE) AND ((EProcessVariables.PicAlpha_HoldingWorkpiece = FALSE) AND ((EProcessVariables.PicAlpha_CylinderRetracted = TRUE) AND ((EProcessVariables.PAC_WPAtStart = FALSE) AND ((EProcessVariables.SSC_ProductType_1 = 0) AND (EProcessVariables.SSC_ProductType_2 = 0)))))
	m_compExpr127: ComparisonExpression(EProcessVariables.PicAlpha_AtPos3, EComparisonType.equals, EDataType.binary, TRUE, 0, '', TRUE);
	m_compExpr129: ComparisonExpression(EProcessVariables.PicAlpha_HoldingWorkpiece, EComparisonType.equals, EDataType.binary, FALSE, 0, '', TRUE);
	m_compExpr131: ComparisonExpression(EProcessVariables.PicAlpha_CylinderRetracted, EComparisonType.equals, EDataType.binary, TRUE, 0, '', TRUE);
	m_compExpr133: ComparisonExpression(EProcessVariables.PAC_WPAtStart, EComparisonType.equals, EDataType.binary, FALSE, 0, '', TRUE);
	m_compExpr135: ComparisonExpression(EProcessVariables.SSC_ProductType_1, EComparisonType.equals, EDataType.numeric, FALSE, 0, '', TRUE);
	m_compExpr137: ComparisonExpression(EProcessVariables.SSC_ProductType_2, EComparisonType.equals, EDataType.numeric, FALSE, 0, '', TRUE);
	m_boolExpr138: BoolExpression(m_compExpr135, EBoolOperation.and_op, m_compExpr137);
	m_boolExpr139: BoolExpression(m_compExpr133, EBoolOperation.and_op, m_boolExpr138);
	m_boolExpr140: BoolExpression(m_compExpr131, EBoolOperation.and_op, m_boolExpr139);
	m_boolExpr141: BoolExpression(m_compExpr129, EBoolOperation.and_op, m_boolExpr140);
	m_precondition: BoolExpression(m_compExpr127, EBoolOperation.and_op, m_boolExpr141);
	
	// EProcessVariables.PAC_WPAtEnd = FALSE
	m_postcondition: ComparisonExpression(EProcessVariables.PAC_WPAtEnd, EComparisonType.equals, EDataType.binary, FALSE, 0, '', TRUE);
	
	m_timer : TON;
END_VAR

SUPER^();

METHOD PROTECTED  AtTarget : BOOL
VAR_INPUT
END_VAR
//AtTarget := FALSE;
IF NOT m_ptrPAC^.WPAtEnd THEN
	m_timer(IN := TRUE, PT := T#1500MS);
	IF m_timer.Q THEN
		m_timer(IN := FALSE);
		m_ptrPAC^.METH_ResetWPNumberAtPAC();
		AtTarget := TRUE;
	END_IF
END_IF
END_METHOD

METHOD PROTECTED EjectOperation : BOOL
VAR_INPUT
END_VAR
EjectOperation := TRUE;
END_METHOD

METHOD FB_init : BOOL
VAR_INPUT
	bInitRetains : BOOL; // if TRUE, the retain variables are initialized (warm start / cold start)
	bInCopyCode : BOOL;  // if TRUE, the instance afterwards gets moved into the copy code (online change)
	
	i_ptrPAC: POINTER TO PicAlphaConveyor;
END_VAR
m_ptrPAC := i_ptrPAC;

m_id := EPrimitives.PAC_TransferWorkpieceTo_SSC;
m_timeout := T#200S;

Precondition := m_precondition;
Postcondition := m_postcondition;
END_METHOD

END_FUNCTION_BLOCK

// ---- 03_ControlPrimitives/Conveyor/RFC/RFC_MoveWorkpiece_Base.TcPOU
FUNCTION_BLOCK ABSTRACT RFC_MoveWorkpiece_Base EXTENDS ControlPrimitiveBase
VAR_INPUT
END_VAR
VAR_OUTPUT
END_VAR
VAR
	m_ptrRFC: POINTER TO RefeedingConveyor;
	
	m_step: INT := 0;
END_VAR

SUPER^();

METHOD  Abort : BOOL
VAR_INPUT
END_VAR
m_ptrRFC^.METH_ConveyorStop();
m_ptrRFC^.METH_Switch_Retract();
Abort := TRUE;
END_METHOD

METHOD PROTECTED ABSTRACT AtTarget : BOOL
VAR_INPUT
END_VAR
END_METHOD

(* Execution logic of this Control Primitive. *)
METHOD PROTECTED ExecuteInternal : BOOL
VAR_INPUT
	i_params: ParameterSet;
END_VAR
CASE m_step OF
	0: // to target	
	IF NOT AtTarget() THEN
		m_ptrRFC^.METH_ConveyorForward();
		m_step := 1;
	END_IF
		
	1:
	IF AtTarget() THEN
		m_ptrRFC^.METH_ConveyorStop();
		//m_ptrPAC^.METH_Switch_Extend();
		m_step := 0;
		ExecuteInternal := TRUE;
	END_IF
		
END_CASE
END_METHOD

END_FUNCTION_BLOCK

// ---- 05_HardwareControl/EquipmentModule/Conveyors/RefeedingConveyor.TcPOU
FUNCTION_BLOCK RefeedingConveyor EXTENDS Conveyor
VAR_INPUT
END_VAR
VAR_OUTPUT
END_VAR
VAR
	//Sensors
	m_PresencesensorStart : PresenceSensor;
	m_PresencesensorEnd : PresenceSensor;
	
	//Pusher
	m_Switch : Switch;
END_VAR

METHOD METH_Switch_Extend : BOOL
VAR_INPUT
END_VAR
m_Switch.METH_Extend();
END_METHOD

METHOD METH_Switch_Retract : BOOL
VAR_INPUT
END_VAR
m_Switch.METH_Retract();
END_METHOD

PROPERTY WPAtEnd : BOOL
GET
WPAtEnd := m_PresencesensorEnd.Value;
END_GET
END_PROPERTY

PROPERTY WPAtStart : BOOL
GET
WPAtStart := m_PresencesensorStart.Value;
END_GET
END_PROPERTY

END_FUNCTION_BLOCK

// ---- 03_ControlPrimitives/Conveyor/RFC/RFC_TransferWorkpieceTo_LSC.TcPOU
FUNCTION_BLOCK RFC_TransferWorkpieceTo_LSC EXTENDS RFC_MoveWorkpiece_Base
VAR_INPUT
END_VAR
VAR_OUTPUT
END_VAR
VAR
	// (EProcessVariables.LSC_ProductType = 0) AND ((EProcessVariables.RFC_WPAtEnd = TRUE) AND ((EProcessVariables.Crane_AtLSC = FALSE) OR ((EProcessVariables.Crane_AtLSC = TRUE) AND ((EProcessVariables.Crane_CylinderRetracted = TRUE) AND (EProcessVariables.Crane_HoldingWorkpiece = FALSE)))))
	m_compExpr203: ComparisonExpression(EProcessVariables.LSC_ProductType, EComparisonType.equals, EDataType.numeric, FALSE, 0, '', TRUE);
	m_compExpr205: ComparisonExpression(EProcessVariables.RFC_WPAtEnd, EComparisonType.equals, EDataType.binary, TRUE, 0, '', TRUE);
	m_compExpr207: ComparisonExpression(EProcessVariables.Crane_AtLSC, EComparisonType.equals, EDataType.binary, FALSE, 0, '', TRUE);
	m_compExpr209: ComparisonExpression(EProcessVariables.Crane_AtLSC, EComparisonType.equals, EDataType.binary, TRUE, 0, '', TRUE);
	m_compExpr211: ComparisonExpression(EProcessVariables.Crane_CylinderRetracted, EComparisonType.equals, EDataType.binary, TRUE, 0, '', TRUE);
	m_compExpr213: ComparisonExpression(EProcessVariables.Crane_HoldingWorkpiece, EComparisonType.equals, EDataType.binary, FALSE, 0, '', TRUE);
	m_boolExpr214: BoolExpression(m_compExpr211, EBoolOperation.and_op, m_compExpr213);
	m_boolExpr215: BoolExpression(m_compExpr209, EBoolOperation.and_op, m_boolExpr214);
	m_boolExpr216: BoolExpression(m_compExpr207, EBoolOperation.or_op, m_boolExpr215);
	m_boolExpr217: BoolExpression(m_compExpr205, EBoolOperation.and_op, m_boolExpr216);
	m_precondition: BoolExpression(m_compExpr203, EBoolOperation.and_op, m_boolExpr217);
	
	// EProcessVariables.RFC_SwitchRetracted = TRUE
	m_postcondition: ComparisonExpression(EProcessVariables.RFC_SwitchRetracted, EComparisonType.equals, EDataType.binary, TRUE, 0, '', TRUE);
		
	m_case: UINT := 0;
	m_timer: TON;
END_VAR

SUPER^();

METHOD PROTECTED  AtTarget : BOOL
VAR_INPUT
END_VAR
AtTarget := FALSE;

CASE m_case OF
	0:
		m_ptrRFC^.METH_Switch_Extend();
		m_timer(IN := TRUE, PT := T#200MS);
		IF m_timer.Q THEN
			m_case := 1;
			m_timer(IN := FALSE);
		END_IF
	
	1:
		m_ptrRFC^.METH_Switch_Retract();
		m_timer(IN := TRUE, PT := T#1000MS);
		IF m_timer.Q THEN
			m_case := 0;
			m_timer(IN := FALSE);
			AtTarget := TRUE;
		END_IF
	
END_CASE
END_METHOD

METHOD FB_init : BOOL
VAR_INPUT
	bInitRetains : BOOL; // if TRUE, the retain variables are initialized (warm start / cold start)
	bInCopyCode : BOOL;  // if TRUE, the instance afterwards gets moved into the copy code (online change)
	
	i_ptrRFC: POINTER TO RefeedingConveyor;
END_VAR
m_ptrRFC := i_ptrRFC;

m_id := EPrimitives.RFC_TransferWorkpieceTo_LSC;
m_timeout := T#200S;

Precondition := m_precondition;
Postcondition := m_postcondition;
END_METHOD

END_FUNCTION_BLOCK

// ---- 03_ControlPrimitives/Conveyor/RFC/RFC_TransferWorkpieceTo_PSEnd.TcPOU
FUNCTION_BLOCK RFC_TransferWorkpieceTo_PSEnd EXTENDS RFC_MoveWorkpiece_Base
VAR_INPUT
END_VAR
VAR_OUTPUT
END_VAR
VAR
	// EProcessVariables.SSC_WPAtEnd = TRUE
	m_precondition: ComparisonExpression(EProcessVariables.SSC_WPAtEnd, EComparisonType.equals, EDataType.binary, TRUE, 0, '', TRUE);
	
	// EProcessVariables.RFC_WPAtEnd = TRUE
	m_postcondition: ComparisonExpression(EProcessVariables.RFC_WPAtEnd, EComparisonType.equals, EDataType.binary, TRUE, 0, '', TRUE);
END_VAR

SUPER^();

METHOD PROTECTED  AtTarget : BOOL
VAR_INPUT
END_VAR
AtTarget := FALSE;
IF m_ptrRFC^.WPAtEnd THEN
	AtTarget := TRUE;
END_IF
END_METHOD

METHOD FB_init : BOOL
VAR_INPUT
	bInitRetains : BOOL; // if TRUE, the retain variables are initialized (warm start / cold start)
	bInCopyCode : BOOL;  // if TRUE, the instance afterwards gets moved into the copy code (online change)
	
	i_ptrRFC: POINTER TO RefeedingConveyor;
END_VAR
m_ptrRFC := i_ptrRFC;

m_id := EPrimitives.RFC_TransferWorkpieceTo_PSEnd;
m_timeout := T#200S;

Precondition := m_precondition;
Postcondition := m_postcondition;
END_METHOD

END_FUNCTION_BLOCK

// ---- 03_ControlPrimitives/Conveyor/SSC/SSC_MoveWorkpiece_Base.TcPOU
FUNCTION_BLOCK ABSTRACT SSC_MoveWorkpiece_Base EXTENDS ControlPrimitiveBase
VAR_INPUT
END_VAR
VAR_OUTPUT
END_VAR
VAR
	m_ptrSSC: POINTER TO SmallSortingConveyor;
	
	m_step: INT := 0;
	m_TurnSwitch : BOOL;
END_VAR

SUPER^();

METHOD  Abort : BOOL
VAR_INPUT
END_VAR
m_ptrSSC^.METH_ConveyorStop();
m_ptrSSC^.METH_Switch_Retract();
Abort := TRUE;
END_METHOD

METHOD PROTECTED ABSTRACT AtTarget : BOOL
VAR_INPUT
END_VAR
END_METHOD

(* Execution logic of this Control Primitive. *)
METHOD PROTECTED ExecuteInternal : BOOL
VAR_INPUT
	i_params: ParameterSet;
END_VAR
CASE m_step OF
	0: // to target	
	IF NOT AtTarget() THEN
		m_ptrSSC^.METH_ConveyorForward();
		IF m_TurnSwitch THEN
			m_ptrSSC^.METH_Switch_Extend();
		END_IF
		m_step := 1;
	END_IF
		
	1:
	IF AtTarget() THEN
		m_ptrSSC^.METH_ConveyorStop();
		IF NOT m_TurnSwitch THEN
			m_ptrSSC^.METH_Switch_Retract();
		END_IF
		m_step := 0;
		ExecuteInternal := TRUE;
	END_IF
		
END_CASE
END_METHOD

END_FUNCTION_BLOCK

// ---- 05_HardwareControl/EquipmentModule/Conveyors/SmallSortingConveyor.TcPOU
FUNCTION_BLOCK SmallSortingConveyor EXTENDS Conveyor
VAR_INPUT
END_VAR
VAR_OUTPUT
END_VAR
VAR
	//Sensors
	m_PresencesensorStart : PresenceSensor;
	m_PresencesensorEnd : PresenceSensor;
	m_Opticalsensor : OpticalSensor;
	m_Inductivesensor : InductiveSensor;
	
	//Ramps
	m_Ramp : Ramp;
	
	//Pusher
	m_Switch : Switch;
END_VAR

PROPERTY LightWPAtMid : BOOL
GET
LightWPAtMid := m_Opticalsensor.Value;
END_GET
END_PROPERTY

PROPERTY MetalWPAtMid : BOOL
GET
MetalWPAtMid := m_Inductivesensor.Value;
END_GET
END_PROPERTY

METHOD METH_Switch_Extend : BOOL
VAR_INPUT
END_VAR
m_Switch.METH_Extend();
END_METHOD

METHOD METH_Switch_Retract : BOOL
VAR_INPUT
END_VAR
m_Switch.METH_Retract();
END_METHOD

PROPERTY WPAtEnd : BOOL
GET
WPAtEnd := m_PresencesensorEnd.Value;
END_GET
END_PROPERTY

PROPERTY WPAtRampEnd : BOOL
GET
WPAtRampEnd := m_Ramp.m_presenceSensorRampFull.Value;
END_GET
END_PROPERTY

PROPERTY WPAtStart : BOOL
GET
WPAtStart := m_PresencesensorStart.Value;
END_GET
END_PROPERTY

END_FUNCTION_BLOCK

// ---- 03_ControlPrimitives/Conveyor/SSC/SSC_TransferWorkpieceTo_PSStart.TcPOU
FUNCTION_BLOCK SSC_TransferWorkpieceTo_PSStart EXTENDS SSC_MoveWorkpiece_Base
VAR_INPUT
END_VAR
VAR_OUTPUT
END_VAR
VAR
	// (EProcessVariables.PicAlpha_HoldingWorkpiece = FALSE) AND ((EProcessVariables.PicAlpha_CylinderRetracted = TRUE) AND (EProcessVariables.PicAlpha_AtPos4 = TRUE))
	m_compExpr226: ComparisonExpression(EProcessVariables.PicAlpha_HoldingWorkpiece, EComparisonType.equals, EDataType.binary, FALSE, 0, '', TRUE);
	m_compExpr228: ComparisonExpression(EProcessVariables.PicAlpha_CylinderRetracted, EComparisonType.equals, EDataType.binary, TRUE, 0, '', TRUE);
	m_compExpr230: ComparisonExpression(EProcessVariables.PicAlpha_AtPos4, EComparisonType.equals, EDataType.binary, TRUE, 0, '', TRUE);
	m_boolExpr231: BoolExpression(m_compExpr228, EBoolOperation.and_op, m_compExpr230);
	m_precondition: BoolExpression(m_compExpr226, EBoolOperation.and_op, m_boolExpr231);
	
	// EProcessVariables.SSC_WPAtStart = TRUE
	m_postcondition: ComparisonExpression(EProcessVariables.SSC_WPAtStart, EComparisonType.equals, EDataType.binary, TRUE, 0, '', TRUE);
END_VAR

SUPER^();

METHOD PROTECTED  AtTarget : BOOL
VAR_INPUT
END_VAR
//AtTarget := FALSE;
IF m_ptrSSC^.WPAtStart THEN
	AtTarget := TRUE;
END_IF
END_METHOD

METHOD FB_init : BOOL
VAR_INPUT
	bInitRetains : BOOL; // if TRUE, the retain variables are initialized (warm start / cold start)
	bInCopyCode : BOOL;  // if TRUE, the instance afterwards gets moved into the copy code (online change)
	
	i_ptrSSC: POINTER TO SmallSortingConveyor;
END_VAR
m_ptrSSC := i_ptrSSC;

m_id := EPrimitives.SSC_TransferWorkpieceTo_PSStart;
m_timeout := T#200S;

Precondition := m_precondition;
Postcondition := m_postcondition;
END_METHOD

END_FUNCTION_BLOCK

// ---- 03_ControlPrimitives/Conveyor/SSC/SSC_TransferWorkpieceTo_RampEnd.TcPOU
FUNCTION_BLOCK SSC_TransferWorkpieceTo_RampEnd EXTENDS SSC_MoveWorkpiece_Base
VAR_INPUT
END_VAR
VAR_OUTPUT
END_VAR
VAR
	// (EProcessVariables.PicAlpha_AtPos3 = TRUE) AND ((EProcessVariables.PicAlpha_HoldingWorkpiece = FALSE) AND (EProcessVariables.PicAlpha_CylinderExtended = FALSE))
	m_compExpr233: ComparisonExpression(EProcessVariables.PicAlpha_AtPos3, EComparisonType.equals, EDataType.binary, TRUE, 0, '', TRUE);
	m_compExpr235: ComparisonExpression(EProcessVariables.PicAlpha_HoldingWorkpiece, EComparisonType.equals, EDataType.binary, FALSE, 0, '', TRUE);
	m_compExpr237: ComparisonExpression(EProcessVariables.PicAlpha_CylinderExtended, EComparisonType.equals, EDataType.binary, FALSE, 0, '', TRUE);
	m_boolExpr238: BoolExpression(m_compExpr235, EBoolOperation.and_op, m_compExpr237);
	m_precondition: BoolExpression(m_compExpr233, EBoolOperation.and_op, m_boolExpr238);
	
	// TRUE
	m_postcondition: ValueExpression(EDataType.binary, TRUE, 0, '', TRUE);
	
	m_timer: TON;
	m_passby : BOOL;
END_VAR

SUPER^();

METHOD PROTECTED  AtTarget : BOOL
VAR_INPUT
END_VAR

IF m_ptrSSC^.WPAtRampEnd THEN
	m_passby := TRUE;
END_IF

IF m_passby THEN
	m_timer(IN := TRUE, PT := T#200MS);
	IF m_timer.Q THEN
		m_timer(IN := FALSE);
		m_passby := FALSE;
		AtTarget := TRUE;
	END_IF
END_IF
END_METHOD

METHOD FB_init : BOOL
VAR_INPUT
	bInitRetains : BOOL; // if TRUE, the retain variables are initialized (warm start / cold start)
	bInCopyCode : BOOL;  // if TRUE, the instance afterwards gets moved into the copy code (online change)
	
	i_ptrSSC: POINTER TO SmallSortingConveyor;
END_VAR
m_ptrSSC := i_ptrSSC;

m_id := EPrimitives.SSC_TransferWorkpieceTo_RampEnd;
m_timeout := T#200S;

Precondition := m_precondition;
Postcondition := m_postcondition;
END_METHOD

END_FUNCTION_BLOCK

// ---- 03_ControlPrimitives/Conveyor/SSC/SSC_TransferWorkpieceTo_RFC.TcPOU
FUNCTION_BLOCK SSC_TransferWorkpieceTo_RFC EXTENDS SSC_MoveWorkpiece_Base
VAR_INPUT
END_VAR
VAR_OUTPUT
END_VAR
VAR
	// (EProcessVariables.PAC_WPAtStart = FALSE) AND ((EProcessVariables.PAC_WPAtEnd = TRUE) AND ((EProcessVariables.PicAlpha_HoldingWorkpiece = FALSE) AND ((EProcessVariables.PicAlpha_CylinderRetracted = TRUE) AND ((EProcessVariables.RFC_ProductType_1 = 0) AND (EProcessVariables.RFC_ProductType_2 = 0)))))
	m_compExpr242: ComparisonExpression(EProcessVariables.PAC_WPAtStart, EComparisonType.equals, EDataType.binary, FALSE, 0, '', TRUE);
	m_compExpr244: ComparisonExpression(EProcessVariables.PAC_WPAtEnd, EComparisonType.equals, EDataType.binary, TRUE, 0, '', TRUE);
	m_compExpr246: ComparisonExpression(EProcessVariables.PicAlpha_HoldingWorkpiece, EComparisonType.equals, EDataType.binary, FALSE, 0, '', TRUE);
	m_compExpr248: ComparisonExpression(EProcessVariables.PicAlpha_CylinderRetracted, EComparisonType.equals, EDataType.binary, TRUE, 0, '', TRUE);
	m_compExpr250: ComparisonExpression(EProcessVariables.RFC_ProductType_1, EComparisonType.equals, EDataType.numeric, FALSE, 0, '', TRUE);
	m_compExpr252: ComparisonExpression(EProcessVariables.RFC_ProductType_2, EComparisonType.equals, EDataType.numeric, FALSE, 0, '', TRUE);
	m_boolExpr253: BoolExpression(m_compExpr250, EBoolOperation.and_op, m_compExpr252);
	m_boolExpr254: BoolExpression(m_compExpr248, EBoolOperation.and_op, m_boolExpr253);
	m_boolExpr255: BoolExpression(m_compExpr246, EBoolOperation.and_op, m_boolExpr254);
	m_boolExpr256: BoolExpression(m_compExpr244, EBoolOperation.and_op, m_boolExpr255);
	m_precondition: BoolExpression(m_compExpr242, EBoolOperation.and_op, m_boolExpr256);
	
	// TRUE
	m_postcondition: ValueExpression(EDataType.binary, TRUE, 0, '', TRUE);
	
	m_timer : TON;
END_VAR

SUPER^();

METHOD PROTECTED  AtTarget : BOOL
VAR_INPUT
END_VAR
//AtTarget := FALSE;
m_TurnSwitch := TRUE;


IF NOT m_ptrSSC^.WPAtRampEnd THEN
	m_timer(IN := TRUE, PT := T#3500MS);
	IF m_timer.Q THEN
		m_timer(IN := FALSE);
		m_TurnSwitch := FALSE;
		AtTarget := TRUE;
	END_IF
END_IF
END_METHOD

METHOD FB_init : BOOL
VAR_INPUT
	bInitRetains : BOOL; // if TRUE, the retain variables are initialized (warm start / cold start)
	bInCopyCode : BOOL;  // if TRUE, the instance afterwards gets moved into the copy code (online change)
	
	i_ptrSSC: POINTER TO SmallSortingConveyor;
END_VAR
m_ptrSSC := i_ptrSSC;

m_id := EPrimitives.SSC_TransferWorkpieceTo_RFC;
m_timeout := T#200S;

Precondition := m_precondition;
Postcondition := m_postcondition;
END_METHOD

END_FUNCTION_BLOCK

// ---- 03_ControlPrimitives/Generic/Delay.TcPOU
FUNCTION_BLOCK Delay EXTENDS ControlPrimitiveBase
VAR_INPUT
END_VAR
VAR_OUTPUT
END_VAR
VAR
	m_precondition: ValueExpression(EDataType.binary, TRUE, 0, '', TRUE);
	m_postcondition: ValueExpression(EDataType.binary, TRUE, 0, '', TRUE);
	
	m_ton: TON;
END_VAR

SUPER^();

METHOD Abort : BOOL
VAR_INPUT
END_VAR
Abort := TRUE;
END_METHOD

(* Execution logic of this Control Primitive. *)
METHOD PROTECTED ExecuteInternal : BOOL
VAR_INPUT
	(*
	 * ms: UINT
	 *)
	i_params: ParameterSet;
END_VAR
VAR
	m_msVal: SNamedValue;
END_VAR
m_msVal := i_params.Retrieve('ms');
m_ton(IN := TRUE, PT := LREAL_TO_TIME(m_msVal.Value.Numeric));
IF m_ton.Q THEN
	m_ton(IN := FALSE);
	ExecuteInternal := TRUE;
ELSE
	ExecuteInternal := FALSE;
END_IF
END_METHOD

METHOD FB_init : BOOL
VAR_INPUT
	bInitRetains : BOOL; // if TRUE, the retain variables are initialized (warm start / cold start)
	bInCopyCode : BOOL;  // if TRUE, the instance afterwards gets moved into the copy code (online change)
END_VAR
m_id := EPrimitives.Gen_Delay;
m_timeout := T#99999S;
m_paramDefinition := 'ms:UINT;';

Precondition := m_precondition;
Postcondition := m_postcondition;
END_METHOD

END_FUNCTION_BLOCK

// ---- 03_ControlPrimitives/Generic/ForceProcessVariable.TcPOU
FUNCTION_BLOCK ForceProcessVariable EXTENDS ControlPrimitiveBase
VAR_INPUT
END_VAR
VAR_OUTPUT
END_VAR
VAR
	m_precondition: ValueExpression(EDataType.binary, TRUE, 0, '', TRUE);
	m_postcondition: ValueExpression(EDataType.binary, TRUE, 0, '', TRUE);
END_VAR

SUPER^();

METHOD Abort : BOOL
END_METHOD

(* Execution logic of this Control Primitive. *)
METHOD PROTECTED ExecuteInternal : BOOL
VAR_INPUT
	i_params	: Resi4MPM.ParameterSet;
END_VAR
VAR
	namedVal: SNamedValue;
	varId: UINT;
	dType: EDataType;
END_VAR
ExecuteInternal := FALSE;

namedVal := i_params.Retrieve('variable_id');
varId := LREAL_TO_UINT(namedVal.Value.Numeric);

namedVal := i_params.Retrieve('type');
dType := LREAL_TO_USINT(namedVal.Value.Numeric);
CASE dType OF
	EDataType.binary:
		namedVal := i_params.Retrieve('bool_val');
		THIS^.m_st^.PtrProcessState^.UpdateState_Binary(varId, namedVal.Value.Binary, TRUE);
		ExecuteInternal := TRUE;
	
	EDataType.numeric:
		namedVal := i_params.Retrieve('num_val');
		THIS^.m_st^.PtrProcessState^.UpdateState_Numeric(varId, namedVal.Value.Numeric, TRUE);
		ExecuteInternal := TRUE;
	
	EDataType.string_t:
		namedVal := i_params.Retrieve('string_val');
		THIS^.m_st^.PtrProcessState^.UpdateState_String(varId, namedVal.Value.String_t, TRUE);
		ExecuteInternal := TRUE;
	
	ELSE
		RETURN;
END_CASE
END_METHOD

//FB_Init is always available implicitly and it is used primarily for initialization.
//The return value is not evaluated. For a specific influence, you can also declare the
//methods explicitly and provide additional code there with the standard initialization
//code. You can evaluate the return value.
METHOD FB_Init: BOOL
VAR_INPUT
    bInitRetains: BOOL; // TRUE: the retain variables are initialized (reset warm / reset cold)
    bInCopyCode: BOOL;  // TRUE: the instance will be copied to the copy code afterward (online change)
	
	i_id: UINT;
END_VAR
m_id := i_id;
m_timeout := T#5S;
m_paramDefinition := 'variable_id:UINT;type:EDataType;bool_val:BOOL;num_val:LREAL;string_val:STRING;';

Precondition := m_precondition;
Postcondition := m_postcondition;
END_METHOD

END_FUNCTION_BLOCK

// ---- 03_ControlPrimitives/Generic/IndicateActivity.TcPOU
FUNCTION_BLOCK IndicateActivity EXTENDS ControlPrimitiveBase
VAR
	m_precondition: ValueExpression(EDataType.binary, TRUE, 0, '', TRUE);
// 	m_postcondition: ValueExpression(EDataType.binary, TRUE, 0, '', TRUE);
	m_postcondition: ComparisonExpression(EProcessVariables.LSC_RampEndWPCount, EComparisonType.greater, EDataType.numeric, FALSE, 0, '', TRUE);
	m_ptrIndic: POINTER TO ActivityIndicator;
	
	m_execTon: TON;
	m_blinkTon: TON;
END_VAR

SUPER^();

METHOD Abort : BOOL
VAR_INPUT
END_VAR
Abort := TRUE;
END_METHOD

(* Execution logic of this Control Primitive. *)
METHOD PROTECTED ExecuteInternal : BOOL
VAR_INPUT
	i_params	: Resi4MPM.ParameterSet;
END_VAR
VAR
	m_val: SNamedValue;
	m_dur: TIME;
END_VAR
m_val := i_params.Retrieve('duration_ms');
m_dur := LREAL_TO_TIME(m_val.Value.Numeric);

m_ptrIndic^.ResetDoneSignal();
ExecuteInternal := FALSE;
m_execTon(IN := TRUE, PT := m_dur);

IF m_execTon.Q THEN
	ExecuteInternal := TRUE;
	m_ptrIndic^.SetDoneSignal();
	m_execTon(IN := FALSE);
ELSE
	// "blink" the activity indicator
	m_blinkTon(IN := TRUE, PT := T#200MS);
	IF m_blinkTon.Q THEN
		m_ptrIndic^.FlipIndicator();
		m_blinkTon(IN := FALSE);
	END_IF
END_IF
END_METHOD

//FB_Init is always available implicitly and it is used primarily for initialization.
//The return value is not evaluated. For a specific influence, you can also declare the
//methods explicitly and provide additional code there with the standard initialization
//code. You can evaluate the return value.
METHOD FB_Init: BOOL
VAR_INPUT
    bInitRetains: BOOL; // TRUE: the retain variables are initialized (reset warm / reset cold)
    bInCopyCode: BOOL;  // TRUE: the instance will be copied to the copy code afterward (online change)
	
	i_id: UINT;
	i_ptrIndicator: POINTER TO ActivityIndicator;
END_VAR
m_id := i_id;
m_timeout := T#5S;
m_paramDefinition := 'duration_ms:UINT;';

Precondition := m_precondition;
Postcondition := m_postcondition;

m_ptrIndic := i_ptrIndicator;
END_METHOD

END_FUNCTION_BLOCK

// ---- 05_HardwareControl/ControlModule/Gen/ActivityIndicator.TcPOU
FUNCTION_BLOCK ActivityIndicator EXTENDS HardwareObservationBase
VAR_INPUT
END_VAR
VAR_OUTPUT
END_VAR
VAR
	DO_indic AT%Q*: BOOL;
	
	
	m_sigVar: UINT;
	m_sigState: BOOL;
END_VAR

//FB_Init is always available implicitly and it is used primarily for initialization.
//The return value is not evaluated. For a specific influence, you can also declare the
//methods explicitly and provide additional code there with the standard initialization
//code. You can evaluate the return value.
METHOD FB_Init: BOOL
VAR_INPUT
    bInitRetains: BOOL; // TRUE: the retain variables are initialized (reset warm / reset cold)
    bInCopyCode: BOOL;  // TRUE: the instance will be copied to the copy code afterward (online change)
	
	i_signalProcVar: UINT;
END_VAR
m_sigVar := i_signalProcVar;
END_METHOD

METHOD FlipIndicator : BOOL
VAR_INPUT
END_VAR
m_sigState := FALSE;
DO_indic := NOT DO_indic;
END_METHOD

METHOD  ResetDefinition : BOOL
VAR_INPUT
END_VAR
m_sigState := TRUE;
END_METHOD

METHOD ResetDoneSignal : BOOL
IF m_sigVar = 0 THEN
	ResetDoneSignal := FALSE;
ELSE
	m_sigState  := FALSE;
	ResetDoneSignal := TRUE;
	DO_indic := FALSE;
END_IF
END_METHOD

(*
	Sets the global variable for the "Done" signal to TRUE.
	WIll be reset FlipIndicator is called the next time.
*)
METHOD SetDoneSignal : BOOL
IF m_sigVar = 0 THEN
	SetDoneSignal := FALSE;
ELSE
	m_sigState  := TRUE;
	SetDoneSignal := TRUE;
	DO_indic := FALSE;
END_IF
END_METHOD

(* Update an instance of ProcessState with the part of the process that can be observed by this Hardware Interface. *)
METHOD UpdateProcessObservation : BOOL
VAR_IN_OUT
	io_processState: ProcessState;
END_VAR
io_processState.UpdateState_Binary(m_sigVar, m_sigState, i_force := TRUE);
io_processState.UpdateState_Defined(m_sigVar, TRUE);
END_METHOD

END_FUNCTION_BLOCK

// ---- 03_ControlPrimitives/Stack/Stack_ProvideWorkpiece.TcPOU
FUNCTION_BLOCK Stack_ProvideWorkpiece EXTENDS ControlPrimitiveBase
VAR_INPUT
END_VAR
VAR_OUTPUT
END_VAR
VAR
	// (EProcessVariables.Stack_WorkpieceAvailable = FALSE) AND ((EProcessVariables.Crane_AtStack = FALSE) OR ((EProcessVariables.Crane_AtStack = TRUE) AND (EProcessVariables.Crane_HoldingWorkpiece = FALSE)))
	m_compExpr260: ComparisonExpression(EProcessVariables.Stack_WorkpieceAvailable, EComparisonType.equals, EDataType.binary, FALSE, 0, '', TRUE);
	m_compExpr262: ComparisonExpression(EProcessVariables.Crane_AtStack, EComparisonType.equals, EDataType.binary, FALSE, 0, '', TRUE);
	m_compExpr264: ComparisonExpression(EProcessVariables.Crane_AtStack, EComparisonType.equals, EDataType.binary, TRUE, 0, '', TRUE);
	m_compExpr266: ComparisonExpression(EProcessVariables.Crane_HoldingWorkpiece, EComparisonType.equals, EDataType.binary, FALSE, 0, '', TRUE);
	m_boolExpr267: BoolExpression(m_compExpr264, EBoolOperation.and_op, m_compExpr266);
	m_boolExpr268: BoolExpression(m_compExpr262, EBoolOperation.or_op, m_boolExpr267);
	m_precondition: BoolExpression(m_compExpr260, EBoolOperation.and_op, m_boolExpr268);
	
	// EProcessVariables.Stack_WorkpieceAvailable = TRUE
	m_postcondition: ComparisonExpression(EProcessVariables.Stack_WorkpieceAvailable, EComparisonType.equals, EDataType.binary, TRUE, 0, '', TRUE);
	
	m_ptrStack: POINTER TO Stack;

	m_step: INT;
END_VAR

SUPER^();

METHOD Abort : BOOL
VAR_INPUT
END_VAR
m_ptrStack^.o_slidingCylinder.METH_Retract();
Abort := TRUE;
END_METHOD

(* Execution logic of this Control Primitive. *)
METHOD PROTECTED  ExecuteInternal : BOOL
VAR_INPUT
	i_params: ParameterSet;
END_VAR
CASE m_step OF
	0: // extend
	m_ptrStack^.o_slidingCylinder.METH_Extend();
	IF m_ptrStack^.o_slidingCylinder.Extended THEN
		m_step := 1;
	END_IF
	
	1: // retract
	m_ptrStack^.o_slidingCylinder.METH_Retract();
	IF m_ptrStack^.o_slidingCylinder.Retracted THEN
		ExecuteInternal := TRUE;
		m_step := 0;
	END_IF
END_CASE
END_METHOD

METHOD FB_init : BOOL
VAR_INPUT
	bInitRetains : BOOL; // if TRUE, the retain variables are initialized (warm start / cold start)
	bInCopyCode : BOOL;  // if TRUE, the instance afterwards gets moved into the copy code (online change)
	
	i_ptrStack: POINTER TO Stack;
END_VAR
m_ptrStack := i_ptrStack;

m_id := EPrimitives.Stack_ProvideWorkpiece;
m_timeout := T#5S;

Precondition := m_precondition;
Postcondition := m_postcondition;
END_METHOD

END_FUNCTION_BLOCK

// ---- 05_HardwareControl/EquipmentModule/Stacks/Stack.TcPOU
FUNCTION_BLOCK Stack
VAR_INPUT
END_VAR
VAR_OUTPUT
	o_slidingCylinder : MonostableCylinder;
END_VAR
VAR
	//Sensors
	m_Presencesensor : PresenceSensor;
	m_Opticalsensor : OpticalSensor;
	m_Inductivesensor : InductiveSensor;
	m_Weightsensor : WeightSensor;
END_VAR

PROPERTY LightWPOnTray : BOOL
GET
LightWPOnTray:=m_Opticalsensor.Value;
END_GET
END_PROPERTY

PROPERTY MetalWPOnTray : BOOL
GET
MetalWPOnTray := m_Inductivesensor.Value;
END_GET
END_PROPERTY

PROPERTY WPOnTray : BOOL
 //REFERENCE TO PresenceSensor
GET
WPOnTray:=m_Presencesensor.Value;
END_GET
END_PROPERTY

PROPERTY WPWeight : INT
GET
WPWeight:=m_Weightsensor.Value;
END_GET
END_PROPERTY

END_FUNCTION_BLOCK

// ---- 05_HardwareControl/ControlModule/Sensors/WeightSensor.TcPOU
FUNCTION_BLOCK WeightSensor IMPLEMENTS ITF_AnalogSensor
VAR_INPUT
END_VAR
VAR_OUTPUT
END_VAR
VAR
	AI_WPWeight AT %I* : INT;
END_VAR

PROPERTY Value : INT
GET
Value := AI_WPWeight;
END_GET
END_PROPERTY

END_FUNCTION_BLOCK

